LIN {X 0,Y 419.877,Z 411.6,A -85,B 0,C 180,E1 9458.97,E2 9458.97} C_VEL
LIN {X 0,Y 420.638,Z 405.188,A -85,B 0,C 180,E1 9462.43,E2 9462.43} C_VEL
LIN {X 0,Y 421.745,Z 393.076,A -85,B 0,C 180,E1 9465.832,E2 9465.832} C_VEL
LIN {X 0,Y 423.274,Z 375.401,A -85,B 0,C 180,E1 9468.881,E2 9468.881} C_VEL
LIN {X 0,Y 424.894,Z 354.463,A -85,B 0,C 180,E1 9471.197,E2 9471.197} C_VEL
LIN {X 0,Y 425.891,Z 330.735,A -85,B 0,C 180,E1 9472.858,E2 9472.858} C_VEL
LIN {X 0,Y 419.501,Z 305.694,A -85,B 0,C 180,E1 9474.153,E2 9474.153} C_VEL
LIN {X 0,Y 417.305,Z 297.81,A -85,B 0,C 180,E1 9474.446,E2 9474.446} C_VEL
LIN {X 0,Y 416.963,Z 297.81,A -85,B 0,C 180,E1 9480.442,E2 9480.442} C_VEL
LIN {X 0,Y 416.972,Z 297.81,A -85,B 0,C 180,E1 9487.211,E2 9487.211} C_VEL
LIN {X 0,Y 416.83,Z 297.81,A -85,B 0,C 180,E1 9493.591,E2 9493.591} C_VEL
LIN {X 0,Y 416.903,Z 297.81,A -85,B 0,C 180,E1 9499.474,E2 9499.474} C_VEL
LIN {X 0,Y 416.902,Z 297.81,A -85,B 0,C 180,E1 9504.594,E2 9504.594} C_VEL
LIN {X 0,Y 417.002,Z 297.81,A -85,B 0,C 180,E1 9511.922,E2 9511.922} C_VEL
LIN {X 0,Y 417.371,Z 297.81,A -85,B 0,C 180,E1 9518.79,E2 9518.79} C_VEL
LIN {X 0,Y 417.453,Z 297.81,A -85,B 0,C 180,E1 9525.329,E2 9525.329} C_VEL
LIN {X 0,Y 417.766,Z 297.81,A -85,B 0,C 180,E1 9531.679,E2 9531.679} C_VEL
LIN {X 0,Y 418.193,Z 297.81,A -85,B 0,C 180,E1 9537.919,E2 9537.919} C_VEL
LIN {X 0,Y 418.002,Z 297.81,A -85,B 0,C 180,E1 9544.128,E2 9544.128} C_VEL
LIN {X 0,Y 417.732,Z 297.81,A -85,B 0,C 180,E1 9550.393,E2 9550.393} C_VEL
LIN {X 0,Y 417.495,Z 297.81,A -85,B 0,C 180,E1 9556.794,E2 9556.794} C_VEL
LIN {X 0,Y 417.298,Z 297.81,A -85,B 0,C 180,E1 9563.426,E2 9563.426} C_VEL
LIN {X 0,Y 417.029,Z 297.81,A -85,B 0,C 180,E1 9570.423,E2 9570.423} C_VEL
LIN {X 0,Y 416.911,Z 297.81,A -85,B 0,C 180,E1 9577.96,E2 9577.96} C_VEL
LIN {X 0,Y 416.867,Z 297.81,A -85,B 0,C 180,E1 9583.616,E2 9583.616} C_VEL
LIN {X 0,Y 416.962,Z 297.81,A -85,B 0,C 180,E1 9589.446,E2 9589.446} C_VEL
LIN {X 0,Y 416.98,Z 297.81,A -85,B 0,C 180,E1 9594.618,E2 9594.618} C_VEL
LIN {X 0,Y 417.197,Z 297.81,A -85,B 0,C 180,E1 9600.595,E2 9600.595} C_VEL
LIN {X 0,Y 430.602,Z 338.236,A -85,B 0,C 180,E1 9602.059,E2 9602.059} C_VEL
LIN {X 0,Y 429.755,Z 375.538,A -85,B 0,C 180,E1 9602.915,E2 9602.915} C_VEL
LIN {X 0,Y 427.343,Z 408.592,A -85,B 0,C 180,E1 9604.471,E2 9604.471} C_VEL
LIN {X 0,Y 424.757,Z 438.385,A -85,B 0,C 180,E1 9606.719,E2 9606.719} C_VEL
LIN {X 0,Y 422.244,Z 465.016,A -85,B 0,C 180,E1 9609.607,E2 9609.607} C_VEL
LIN {X 0,Y 420.814,Z 481.386,A -85,B 0,C 180,E1 9611.972,E2 9611.972} C_VEL
LIN {X 0,Y 419.147,Z 486.865,A -85,B 0,C 180,E1 9612.877,E2 9612.877} C_VEL
LIN {X 0,Y 411.685,Z 500.03,A -85,B 0,C 180,E1 9615.497,E2 9615.497} C_VEL
LIN {X 0,Y 411.541,Z 501.128,A -85,B 0,C 180,E1 9615.76,E2 9615.76} C_VEL
LIN {X 0,Y 411.062,Z 515.83,A -85,B 0,C 180,E1 9619.957,E2 9619.957} C_VEL
LIN {X 0,Y 411.204,Z 524.231,A -85,B 0,C 180,E1 9623.679,E2 9623.679} C_VEL
LIN {X 0,Y 411.473,Z 528.984,A -85,B 0,C 180,E1 9627.898,E2 9627.898} C_VEL
LIN {X 0,Y 411.46,Z 528.901,A -85,B 0,C 180,E1 9632.101,E2 9632.101} C_VEL
LIN {X 0,Y 411.236,Z 524.018,A -85,B 0,C 180,E1 9636.319,E2 9636.319} C_VEL
LIN {X 0,Y 411.131,Z 513.977,A -85,B 0,C 180,E1 9640.574,E2 9640.574} C_VEL
LIN {X 0,Y 411.714,Z 498.169,A -85,B 0,C 180,E1 9644.865,E2 9644.865} C_VEL
LIN {X 0,Y 413.331,Z 476.598,A -85,B 0,C 180,E1 9648.901,E2 9648.901} C_VEL
LIN {X 0,Y 415.903,Z 450.804,A -85,B 0,C 180,E1 9652.327,E2 9652.327} C_VEL
LIN {X 0,Y 418.823,Z 421.694,A -85,B 0,C 180,E1 9655.045,E2 9655.045} C_VEL
LIN {X 0,Y 421.731,Z 389.924,A -85,B 0,C 180,E1 9657.003,E2 9657.003} C_VEL
LIN {X 0,Y 423.6,Z 356.055,A -85,B 0,C 180,E1 9658.183,E2 9658.183} C_VEL
LIN {X 0,Y 423.18,Z 337.903,A -85,B 0,C 180,E1 9658.562,E2 9658.562} C_VEL
LIN {X 0,Y 409.163,Z 297.81,A -85,B 0,C 180,E1 9660.29,E2 9660.29} C_VEL
LIN {X 0,Y 408.961,Z 297.81,A -85,B 0,C 180,E1 9666.183,E2 9666.183} C_VEL
LIN {X 0,Y 408.78,Z 297.81,A -85,B 0,C 180,E1 9672.431,E2 9672.431} C_VEL
LIN {X 0,Y 408.855,Z 297.81,A -85,B 0,C 180,E1 9678.384,E2 9678.384} C_VEL
LIN {X 0,Y 409.002,Z 297.81,A -85,B 0,C 180,E1 9684.259,E2 9684.259} C_VEL
LIN {X 0,Y 409.091,Z 297.81,A -85,B 0,C 180,E1 9691.36,E2 9691.36} C_VEL
LIN {X 0,Y 409.357,Z 297.81,A -85,B 0,C 180,E1 9698.383,E2 9698.383} C_VEL
LIN {X 0,Y 409.454,Z 297.81,A -85,B 0,C 180,E1 9705.063,E2 9705.063} C_VEL
LIN {X 0,Y 409.789,Z 297.81,A -85,B 0,C 180,E1 9711.543,E2 9711.543} C_VEL
LIN {X 0,Y 410.268,Z 297.81,A -85,B 0,C 180,E1 9717.905,E2 9717.905} C_VEL
LIN {X 0,Y 410.042,Z 297.81,A -85,B 0,C 180,E1 9724.234,E2 9724.234} C_VEL
LIN {X 0,Y 409.776,Z 297.81,A -85,B 0,C 180,E1 9730.624,E2 9730.624} C_VEL
LIN {X 0,Y 409.562,Z 297.81,A -85,B 0,C 180,E1 9737.157,E2 9737.157} C_VEL
LIN {X 0,Y 409.296,Z 297.81,A -85,B 0,C 180,E1 9743.941,E2 9743.941} C_VEL
LIN {X 0,Y 409.29,Z 297.81,A -85,B 0,C 180,E1 9749.69,E2 9749.69} C_VEL
LIN {X 0,Y 417.713,Z 325.419,A -85,B 0,C 180,E1 9751.453,E2 9751.453} C_VEL
LIN {X 0,Y 419.879,Z 339.663,A -85,B 0,C 180,E1 9752.561,E2 9752.561} C_VEL
LIN {X 0,Y 417.771,Z 364.033,A -85,B 0,C 180,E1 9754.786,E2 9754.786} C_VEL
LIN {X 0,Y 415.64,Z 383.831,A -85,B 0,C 180,E1 9757.541,E2 9757.541} C_VEL
LIN {X 0,Y 413.839,Z 399.154,A -85,B 0,C 180,E1 9760.783,E2 9760.783} C_VEL
LIN {X 0,Y 412.798,Z 408.597,A -85,B 0,C 180,E1 9764.011,E2 9764.011} C_VEL
LIN {X 0,Y 412.066,Z 413.417,A -85,B 0,C 180,E1 9767.11,E2 9767.11} C_VEL
LIN {X 0,Y 411.741,Z 414.45,A -85,B 0,C 180,E1 9770.344,E2 9770.344} C_VEL
LIN {X 0,Y 412.094,Z 410.619,A -85,B 0,C 180,E1 9774.135,E2 9774.135} C_VEL
LIN {X 0,Y 413.053,Z 400.769,A -85,B 0,C 180,E1 9777.935,E2 9777.935} C_VEL
LIN {X 0,Y 414.439,Z 385.481,A -85,B 0,C 180,E1 9781.372,E2 9781.372} C_VEL
LIN {X 0,Y 416.184,Z 366.055,A -85,B 0,C 180,E1 9784.209,E2 9784.209} C_VEL
LIN {X 0,Y 417.974,Z 342.348,A -85,B 0,C 180,E1 9786.502,E2 9786.502} C_VEL
LIN {X 0,Y 417.684,Z 329.677,A -85,B 0,C 180,E1 9787.428,E2 9787.428} C_VEL
LIN {X 0,Y 410.6,Z 301.996,A -85,B 0,C 180,E1 9789.12,E2 9789.12} C_VEL
LIN {X 0,Y 409.589,Z 297.81,A -85,B 0,C 180,E1 9789.347,E2 9789.347} C_VEL
LIN {X 0,Y 409.484,Z 297.81,A -85,B 0,C 180,E1 9795.052,E2 9795.052} C_VEL
LIN {X 0,Y 409.654,Z 297.81,A -85,B 0,C 180,E1 9797.865,E2 9797.865} C_VEL
LIN {X 0,Y 416.194,Z 326.756,A -85,B 0,C 180,E1 9799.049,E2 9799.049} C_VEL
LIN {X 0,Y 416.462,Z 347.34,A -85,B 0,C 180,E1 9800.353,E2 9800.353} C_VEL
LIN {X 0,Y 415.154,Z 369.979,A -85,B 0,C 180,E1 9802.561,E2 9802.561} C_VEL
LIN {X 0,Y 413.911,Z 388.142,A -85,B 0,C 180,E1 9805.295,E2 9805.295} C_VEL
LIN {X 0,Y 412.857,Z 401.668,A -85,B 0,C 180,E1 9808.43,E2 9808.43} C_VEL
LIN {X 0,Y 412.118,Z 410.765,A -85,B 0,C 180,E1 9812.099,E2 9812.099} C_VEL
LIN {X 0,Y 411.871,Z 413.347,A -85,B 0,C 180,E1 9814.203,E2 9814.203} C_VEL
LIN {X 0,Y 411.774,Z 414.218,A -85,B 0,C 180,E1 9816.312,E2 9816.312} C_VEL
LIN {X 0,Y 412.187,Z 412.205,A -85,B 0,C 180,E1 9819.483,E2 9819.483} C_VEL
LIN {X 0,Y 413.007,Z 404.681,A -85,B 0,C 180,E1 9823.17,E2 9823.17} C_VEL
LIN {X 0,Y 414.429,Z 391.258,A -85,B 0,C 180,E1 9826.664,E2 9826.664} C_VEL
LIN {X 0,Y 415.97,Z 373.143,A -85,B 0,C 180,E1 9829.606,E2 9829.606} C_VEL
LIN {X 0,Y 417.706,Z 350.966,A -85,B 0,C 180,E1 9831.907,E2 9831.907} C_VEL
LIN {X 0,Y 417.787,Z 328.647,A -85,B 0,C 180,E1 9833.411,E2 9833.411} C_VEL
LIN {X 0,Y 410.687,Z 302.83,A -85,B 0,C 180,E1 9834.689,E2 9834.689} C_VEL
LIN {X 0,Y 409.334,Z 297.81,A -85,B 0,C 180,E1 9834.959,E2 9834.959} C_VEL
LIN {X 0,Y 408.972,Z 297.81,A -85,B 0,C 180,E1 9841.908,E2 9841.908} C_VEL
LIN {X 0,Y 409.027,Z 297.81,A -85,B 0,C 180,E1 9846.177,E2 9846.177} C_VEL
LIN {X 0,Y 408.848,Z 297.81,A -85,B 0,C 180,E1 9852.403,E2 9852.403} C_VEL
LIN {X 0,Y 408.864,Z 297.81,A -85,B 0,C 180,E1 9858.35,E2 9858.35} C_VEL
LIN {X 0,Y 408.982,Z 297.81,A -85,B 0,C 180,E1 9864.265,E2 9864.265} C_VEL
LIN {X 0,Y 409.055,Z 297.81,A -85,B 0,C 180,E1 9871.327,E2 9871.327} C_VEL
LIN {X 0,Y 409.393,Z 297.81,A -85,B 0,C 180,E1 9878.356,E2 9878.356} C_VEL
LIN {X 0,Y 409.519,Z 297.81,A -85,B 0,C 180,E1 9885.038,E2 9885.038} C_VEL
LIN {X 0,Y 409.833,Z 297.81,A -85,B 0,C 180,E1 9891.517,E2 9891.517} C_VEL
LIN {X 0,Y 410.279,Z 297.81,A -85,B 0,C 180,E1 9897.879,E2 9897.879} C_VEL
LIN {X 0,Y 410.087,Z 297.81,A -85,B 0,C 180,E1 9904.207,E2 9904.207} C_VEL
LIN {X 0,Y 409.817,Z 297.81,A -85,B 0,C 180,E1 9910.596,E2 9910.596} C_VEL
LIN {X 0,Y 409.549,Z 297.81,A -85,B 0,C 180,E1 9917.13,E2 9917.13} C_VEL
LIN {X 0,Y 409.346,Z 297.81,A -85,B 0,C 180,E1 9923.909,E2 9923.909} C_VEL
LIN {X 0,Y 409.149,Z 297.81,A -85,B 0,C 180,E1 9928.636,E2 9928.636} C_VEL
LIN {X 0,Y 408.984,Z 297.81,A -85,B 0,C 180,E1 9936.166,E2 9936.166} C_VEL
LIN {X 0,Y 408.858,Z 297.81,A -85,B 0,C 180,E1 9942.425,E2 9942.425} C_VEL
LIN {X 0,Y 408.929,Z 297.81,A -85,B 0,C 180,E1 9948.377,E2 9948.377} C_VEL
LIN {X 0,Y 409.073,Z 297.81,A -85,B 0,C 180,E1 9954.227,E2 9954.227} C_VEL
LIN {X 0,Y 409.228,Z 297.81,A -85,B 0,C 180,E1 9960.114,E2 9960.114} C_VEL
LIN {X 0,Y 423.137,Z 339.386,A -85,B 0,C 180,E1 9961.671,E2 9961.671} C_VEL
LIN {X 0,Y 422.345,Z 375.855,A -85,B 0,C 180,E1 9962.552,E2 9962.552} C_VEL
LIN {X 0,Y 419.893,Z 407.972,A -85,B 0,C 180,E1 9964.097,E2 9964.097} C_VEL
LIN {X 0,Y 417.096,Z 437.994,A -85,B 0,C 180,E1 9966.407,E2 9966.407} C_VEL
LIN {X 0,Y 414.411,Z 465.492,A -85,B 0,C 180,E1 9969.483,E2 9969.483} C_VEL
LIN {X 0,Y 412.351,Z 489.264,A -85,B 0,C 180,E1 9973.25,E2 9973.25} C_VEL
LIN {X 0,Y 411.541,Z 501.128,A -85,B 0,C 180,E1 9975.76,E2 9975.76} C_VEL
LIN {X 0,Y 410.124,Z 505.338,A -85,B 0,C 180,E1 9976.814,E2 9976.814} C_VEL
LIN {X 0,Y 403.307,Z 514.812,A -85,B 0,C 180,E1 9979.819,E2 9979.819} C_VEL
LIN {X 0,Y 403.204,Z 515.557,A -85,B 0,C 180,E1 9980.112,E2 9980.112} C_VEL
LIN {X 0,Y 403.449,Z 524.741,A -85,B 0,C 180,E1 9984.634,E2 9984.634} C_VEL
LIN {X 0,Y 403.663,Z 527.883,A -85,B 0,C 180,E1 9987.857,E2 9987.857} C_VEL
LIN {X 0,Y 403.624,Z 527.805,A -85,B 0,C 180,E1 9992.142,E2 9992.142} C_VEL
LIN {X 0,Y 403.373,Z 522.91,A -85,B 0,C 180,E1 9996.443,E2 9996.443} C_VEL
LIN {X 0,Y 403.27,Z 512.845,A -85,B 0,C 180,E1 10000.783,E2 10000.783} C_VEL
LIN {X 0,Y 403.917,Z 497.006,A -85,B 0,C 180,E1 10005.159,E2 10005.159} C_VEL
LIN {X 0,Y 405.654,Z 475.39,A -85,B 0,C 180,E1 10009.273,E2 10009.273} C_VEL
LIN {X 0,Y 408.359,Z 450.086,A -85,B 0,C 180,E1 10012.696,E2 10012.696} C_VEL
LIN {X 0,Y 411.497,Z 420.27,A -85,B 0,C 180,E1 10015.523,E2 10015.523} C_VEL
LIN {X 0,Y 414.479,Z 389.251,A -85,B 0,C 180,E1 10017.457,E2 10017.457} C_VEL
LIN {X 0,Y 416.489,Z 354.953,A -85,B 0,C 180,E1 10018.663,E2 10018.663} C_VEL
LIN {X 0,Y 416.104,Z 339.832,A -85,B 0,C 180,E1 10018.992,E2 10018.992} C_VEL
LIN {X 0,Y 401.893,Z 300.98,A -85,B 0,C 180,E1 10020.724,E2 10020.724} C_VEL
LIN {X 0,Y 401.173,Z 297.81,A -85,B 0,C 180,E1 10020.968,E2 10020.968} C_VEL
LIN {X 0,Y 400.918,Z 297.81,A -85,B 0,C 180,E1 10027.796,E2 10027.796} C_VEL
LIN {X 0,Y 400.891,Z 297.81,A -85,B 0,C 180,E1 10034.359,E2 10034.359} C_VEL
LIN {X 0,Y 400.96,Z 297.81,A -85,B 0,C 180,E1 10040.24,E2 10040.24} C_VEL
LIN {X 0,Y 401.053,Z 297.81,A -85,B 0,C 180,E1 10045.869,E2 10045.869} C_VEL
LIN {X 0,Y 401.226,Z 297.81,A -85,B 0,C 180,E1 10053.186,E2 10053.186} C_VEL
LIN {X 0,Y 401.479,Z 297.81,A -85,B 0,C 180,E1 10060.242,E2 10060.242} C_VEL
LIN {X 0,Y 401.647,Z 297.81,A -85,B 0,C 180,E1 10067.638,E2 10067.638} C_VEL
LIN {X 0,Y 402.101,Z 297.81,A -85,B 0,C 180,E1 10073.549,E2 10073.549} C_VEL
LIN {X 0,Y 402.314,Z 297.81,A -85,B 0,C 180,E1 10080.013,E2 10080.013} C_VEL
LIN {X 0,Y 402.019,Z 297.81,A -85,B 0,C 180,E1 10086.479,E2 10086.479} C_VEL
LIN {X 0,Y 401.819,Z 297.81,A -85,B 0,C 180,E1 10093.036,E2 10093.036} C_VEL
LIN {X 0,Y 401.481,Z 297.81,A -85,B 0,C 180,E1 10100.01,E2 10100.01} C_VEL
LIN {X 0,Y 401.265,Z 297.81,A -85,B 0,C 180,E1 10106.841,E2 10106.841} C_VEL
LIN {X 0,Y 401.343,Z 297.81,A -85,B 0,C 180,E1 10109.099,E2 10109.099} C_VEL
LIN {X 0,Y 410.289,Z 326.49,A -85,B 0,C 180,E1 10111.007,E2 10111.007} C_VEL
LIN {X 0,Y 412.553,Z 341.624,A -85,B 0,C 180,E1 10112.228,E2 10112.228} C_VEL
LIN {X 0,Y 410.347,Z 365.317,A -85,B 0,C 180,E1 10114.463,E2 10114.463} C_VEL
LIN {X 0,Y 408.073,Z 385.161,A -85,B 0,C 180,E1 10117.289,E2 10117.289} C_VEL
LIN {X 0,Y 406.171,Z 400.332,A -85,B 0,C 180,E1 10120.576,E2 10120.576} C_VEL
LIN {X 0,Y 405.048,Z 409.833,A -85,B 0,C 180,E1 10123.913,E2 10123.913} C_VEL
LIN {X 0,Y 404.135,Z 415.11,A -85,B 0,C 180,E1 10127.772,E2 10127.772} C_VEL
LIN {X 0,Y 403.993,Z 414.846,A -85,B 0,C 180,E1 10131.688,E2 10131.688} C_VEL
LIN {X 0,Y 404.503,Z 409.804,A -85,B 0,C 180,E1 10135.182,E2 10135.182} C_VEL
LIN {X 0,Y 405.56,Z 398.95,A -85,B 0,C 180,E1 10138.875,E2 10138.875} C_VEL
LIN {X 0,Y 407.143,Z 382.739,A -85,B 0,C 180,E1 10142.243,E2 10142.243} C_VEL
LIN {X 0,Y 409.085,Z 361.576,A -85,B 0,C 180,E1 10145.114,E2 10145.114} C_VEL
LIN {X 0,Y 410.898,Z 336.576,A -85,B 0,C 180,E1 10147.321,E2 10147.321} C_VEL
LIN {X 0,Y 405.079,Z 310.18,A -85,B 0,C 180,E1 10149.132,E2 10149.132} C_VEL
LIN {X 0,Y 401.661,Z 297.81,A -85,B 0,C 180,E1 10149.818,E2 10149.818} C_VEL
LIN {X 0,Y 401.744,Z 297.81,A -85,B 0,C 180,E1 10157.539,E2 10157.539} C_VEL
LIN {X 0,Y 408.083,Z 325.34,A -85,B 0,C 180,E1 10158.629,E2 10158.629} C_VEL
LIN {X 0,Y 409.223,Z 339.175,A -85,B 0,C 180,E1 10159.443,E2 10159.443} C_VEL
LIN {X 0,Y 408.028,Z 363.678,A -85,B 0,C 180,E1 10161.494,E2 10161.494} C_VEL
LIN {X 0,Y 406.616,Z 383.649,A -85,B 0,C 180,E1 10164.143,E2 10164.143} C_VEL
LIN {X 0,Y 405.407,Z 399.18,A -85,B 0,C 180,E1 10167.334,E2 10167.334} C_VEL
LIN {X 0,Y 404.445,Z 410.014,A -85,B 0,C 180,E1 10171.07,E2 10171.07} C_VEL
LIN {X 0,Y 404.033,Z 414.49,A -85,B 0,C 180,E1 10174.284,E2 10174.284} C_VEL
LIN {X 0,Y 403.981,Z 415.285,A -85,B 0,C 180,E1 10176.435,E2 10176.435} C_VEL
LIN {X 0,Y 404.438,Z 413.177,A -85,B 0,C 180,E1 10179.666,E2 10179.666} C_VEL
LIN {X 0,Y 405.282,Z 405.709,A -85,B 0,C 180,E1 10183.366,E2 10183.366} C_VEL
LIN {X 0,Y 406.69,Z 393.245,A -85,B 0,C 180,E1 10186.712,E2 10186.712} C_VEL
LIN {X 0,Y 408.337,Z 375.967,A -85,B 0,C 180,E1 10189.664,E2 10189.664} C_VEL
LIN {X 0,Y 410.171,Z 354.486,A -85,B 0,C 180,E1 10192.034,E2 10192.034} C_VEL
LIN {X 0,Y 410.55,Z 331.066,A -85,B 0,C 180,E1 10193.692,E2 10193.692} C_VEL
LIN {X 0,Y 403.638,Z 305.412,A -85,B 0,C 180,E1 10195.035,E2 10195.035} C_VEL
LIN {X 0,Y 401.381,Z 297.81,A -85,B 0,C 180,E1 10195.373,E2 10195.373} C_VEL
LIN {X 0,Y 401.095,Z 297.81,A -85,B 0,C 180,E1 10201.784,E2 10201.784} C_VEL
LIN {X 0,Y 400.972,Z 297.81,A -85,B 0,C 180,E1 10207.762,E2 10207.762} C_VEL
LIN {X 0,Y 400.931,Z 297.81,A -85,B 0,C 180,E1 10214.327,E2 10214.327} C_VEL
LIN {X 0,Y 400.94,Z 297.81,A -85,B 0,C 180,E1 10220.203,E2 10220.203} C_VEL
LIN {X 0,Y 401.039,Z 297.81,A -85,B 0,C 180,E1 10225.874,E2 10225.874} C_VEL
LIN {X 0,Y 401.17,Z 297.81,A -85,B 0,C 180,E1 10233.152,E2 10233.152} C_VEL
LIN {X 0,Y 401.54,Z 297.81,A -85,B 0,C 180,E1 10240.216,E2 10240.216} C_VEL
LIN {X 0,Y 401.719,Z 297.81,A -85,B 0,C 180,E1 10247.597,E2 10247.597} C_VEL
LIN {X 0,Y 402.104,Z 297.81,A -85,B 0,C 180,E1 10253.522,E2 10253.522} C_VEL
LIN {X 0,Y 402.387,Z 297.81,A -85,B 0,C 180,E1 10259.987,E2 10259.987} C_VEL
LIN {X 0,Y 402.082,Z 297.81,A -85,B 0,C 180,E1 10266.451,E2 10266.451} C_VEL
LIN {X 0,Y 401.828,Z 297.81,A -85,B 0,C 180,E1 10273.008,E2 10273.008} C_VEL
LIN {X 0,Y 401.512,Z 297.81,A -85,B 0,C 180,E1 10280.019,E2 10280.019} C_VEL
LIN {X 0,Y 401.271,Z 297.81,A -85,B 0,C 180,E1 10286.811,E2 10286.811} C_VEL
LIN {X 0,Y 401.049,Z 297.81,A -85,B 0,C 180,E1 10294.345,E2 10294.345} C_VEL
LIN {X 0,Y 400.913,Z 297.81,A -85,B 0,C 180,E1 10301.167,E2 10301.167} C_VEL
LIN {X 0,Y 400.998,Z 297.81,A -85,B 0,C 180,E1 10307.362,E2 10307.362} C_VEL
LIN {X 0,Y 401.046,Z 297.81,A -85,B 0,C 180,E1 10312.984,E2 10312.984} C_VEL
LIN {X 0,Y 401.245,Z 297.81,A -85,B 0,C 180,E1 10319.635,E2 10319.635} C_VEL
LIN {X 0,Y 415.97,Z 342.223,A -85,B 0,C 180,E1 10321.318,E2 10321.318} C_VEL
LIN {X 0,Y 414.876,Z 376.886,A -85,B 0,C 180,E1 10322.207,E2 10322.207} C_VEL
LIN {X 0,Y 412.313,Z 409.139,A -85,B 0,C 180,E1 10323.827,E2 10323.827} C_VEL
LIN {X 0,Y 409.318,Z 439.73,A -85,B 0,C 180,E1 10326.29,E2 10326.29} C_VEL
LIN {X 0,Y 406.606,Z 465.95,A -85,B 0,C 180,E1 10329.355,E2 10329.355} C_VEL
LIN {X 0,Y 404.461,Z 489.292,A -85,B 0,C 180,E1 10333.193,E2 10333.193} C_VEL
LIN {X 0,Y 403.34,Z 507.849,A -85,B 0,C 180,E1 10337.577,E2 10337.577} C_VEL
LIN {X 0,Y 403.204,Z 515.557,A -85,B 0,C 180,E1 10340.112,E2 10340.112} C_VEL
LIN {X 0,Y 401.968,Z 518.366,A -85,B 0,C 180,E1 10341.282,E2 10341.282} C_VEL
LIN {X 0,Y 395.684,Z 523.681,A -85,B 0,C 180,E1 10344.572,E2 10344.572} C_VEL
LIN {X 0,Y 395.61,Z 524.049,A -85,B 0,C 180,E1 10344.887,E2 10344.887} C_VEL
LIN {X 0,Y 395.831,Z 526.779,A -85,B 0,C 180,E1 10347.815,E2 10347.815} C_VEL
LIN {X 0,Y 395.794,Z 526.71,A -85,B 0,C 180,E1 10352.184,E2 10352.184} C_VEL
LIN {X 0,Y 395.522,Z 521.807,A -85,B 0,C 180,E1 10356.572,E2 10356.572} C_VEL
LIN {X 0,Y 395.403,Z 511.719,A -85,B 0,C 180,E1 10361,E2 10361} C_VEL
LIN {X 0,Y 396.111,Z 495.854,A -85,B 0,C 180,E1 10365.465,E2 10365.465} C_VEL
LIN {X 0,Y 398.024,Z 474.011,A -85,B 0,C 180,E1 10369.692,E2 10369.692} C_VEL
LIN {X 0,Y 400.985,Z 447.763,A -85,B 0,C 180,E1 10373.269,E2 10373.269} C_VEL
LIN {X 0,Y 404.246,Z 418.855,A -85,B 0,C 180,E1 10376.015,E2 10376.015} C_VEL
LIN {X 0,Y 407.442,Z 386.585,A -85,B 0,C 180,E1 10378.022,E2 10378.022} C_VEL
LIN {X 0,Y 409.482,Z 352.456,A -85,B 0,C 180,E1 10379.194,E2 10379.194} C_VEL
LIN {X 0,Y 408.665,Z 340.268,A -85,B 0,C 180,E1 10379.497,E2 10379.497} C_VEL
LIN {X 0,Y 394.4,Z 301.933,A -85,B 0,C 180,E1 10381.297,E2 10381.297} C_VEL
LIN {X 0,Y 393.225,Z 297.81,A -85,B 0,C 180,E1 10381.622,E2 10381.622} C_VEL
LIN {X 0,Y 393.024,Z 297.81,A -85,B 0,C 180,E1 10387.901,E2 10387.901} C_VEL
LIN {X 0,Y 392.964,Z 297.81,A -85,B 0,C 180,E1 10393.725,E2 10393.725} C_VEL
LIN {X 0,Y 393.066,Z 297.81,A -85,B 0,C 180,E1 10400.156,E2 10400.156} C_VEL
LIN {X 0,Y 393.113,Z 297.81,A -85,B 0,C 180,E1 10407.616,E2 10407.616} C_VEL
LIN {X 0,Y 393.354,Z 297.81,A -85,B 0,C 180,E1 10415.054,E2 10415.054} C_VEL
LIN {X 0,Y 393.593,Z 297.81,A -85,B 0,C 180,E1 10422.153,E2 10422.153} C_VEL
LIN {X 0,Y 393.789,Z 297.81,A -85,B 0,C 180,E1 10428.967,E2 10428.967} C_VEL
LIN {X 0,Y 394.221,Z 297.81,A -85,B 0,C 180,E1 10435.623,E2 10435.623} C_VEL
LIN {X 0,Y 394.412,Z 297.81,A -85,B 0,C 180,E1 10440.014,E2 10440.014} C_VEL
LIN {X 0,Y 394.12,Z 297.81,A -85,B 0,C 180,E1 10446.61,E2 10446.61} C_VEL
LIN {X 0,Y 393.874,Z 297.81,A -85,B 0,C 180,E1 10453.304,E2 10453.304} C_VEL
LIN {X 0,Y 393.566,Z 297.81,A -85,B 0,C 180,E1 10460.202,E2 10460.202} C_VEL
LIN {X 0,Y 393.348,Z 297.81,A -85,B 0,C 180,E1 10467.426,E2 10467.426} C_VEL
LIN {X 0,Y 393.447,Z 298.356,A -85,B 0,C 180,E1 10468.51,E2 10468.51} C_VEL
LIN {X 0,Y 402.553,Z 326.374,A -85,B 0,C 180,E1 10470.447,E2 10470.447} C_VEL
LIN {X 0,Y 405.292,Z 343.205,A -85,B 0,C 180,E1 10471.852,E2 10471.852} C_VEL
LIN {X 0,Y 402.88,Z 367.271,A -85,B 0,C 180,E1 10474.2,E2 10474.2} C_VEL
LIN {X 0,Y 400.472,Z 386.904,A -85,B 0,C 180,E1 10477.095,E2 10477.095} C_VEL
LIN {X 0,Y 398.49,Z 401.676,A -85,B 0,C 180,E1 10480.411,E2 10480.411} C_VEL
LIN {X 0,Y 397.304,Z 411.07,A -85,B 0,C 180,E1 10483.811,E2 10483.811} C_VEL
LIN {X 0,Y 396.525,Z 415.487,A -85,B 0,C 180,E1 10486.765,E2 10486.765} C_VEL
LIN {X 0,Y 396.123,Z 416.783,A -85,B 0,C 180,E1 10489.654,E2 10489.654} C_VEL
LIN {X 0,Y 396.317,Z 414.453,A -85,B 0,C 180,E1 10493.116,E2 10493.116} C_VEL
LIN {X 0,Y 397.096,Z 407.305,A -85,B 0,C 180,E1 10496.75,E2 10496.75} C_VEL
LIN {X 0,Y 398.46,Z 393.887,A -85,B 0,C 180,E1 10500.508,E2 10500.508} C_VEL
LIN {X 0,Y 400.32,Z 375.839,A -85,B 0,C 180,E1 10503.712,E2 10503.712} C_VEL
LIN {X 0,Y 402.402,Z 352.061,A -85,B 0,C 180,E1 10506.474,E2 10506.474} C_VEL
LIN {X 0,Y 402.787,Z 333.301,A -85,B 0,C 180,E1 10507.999,E2 10507.999} C_VEL
LIN {X 0,Y 395.759,Z 305.27,A -85,B 0,C 180,E1 10509.862,E2 10509.862} C_VEL
LIN {X 0,Y 393.753,Z 297.81,A -85,B 0,C 180,E1 10510.262,E2 10510.262} C_VEL
LIN {X 0,Y 393.79,Z 297.81,A -85,B 0,C 180,E1 10517.168,E2 10517.168} C_VEL
LIN {X 0,Y 400.508,Z 326.609,A -85,B 0,C 180,E1 10518.343,E2 10518.343} C_VEL
LIN {X 0,Y 401.645,Z 340.367,A -85,B 0,C 180,E1 10519.173,E2 10519.173} C_VEL
LIN {X 0,Y 400.44,Z 364.205,A -85,B 0,C 180,E1 10521.195,E2 10521.195} C_VEL
LIN {X 0,Y 398.88,Z 385.191,A -85,B 0,C 180,E1 10524.029,E2 10524.029} C_VEL
LIN {X 0,Y 397.611,Z 400.552,A -85,B 0,C 180,E1 10527.282,E2 10527.282} C_VEL
LIN {X 0,Y 396.617,Z 411.25,A -85,B 0,C 180,E1 10531.091,E2 10531.091} C_VEL
LIN {X 0,Y 396.199,Z 415.632,A -85,B 0,C 180,E1 10534.369,E2 10534.369} C_VEL
LIN {X 0,Y 396.308,Z 415.898,A -85,B 0,C 180,E1 10538.005,E2 10538.005} C_VEL
LIN {X 0,Y 397.172,Z 410.434,A -85,B 0,C 180,E1 10542.062,E2 10542.062} C_VEL
LIN {X 0,Y 398.399,Z 399.835,A -85,B 0,C 180,E1 10545.657,E2 10545.657} C_VEL
LIN {X 0,Y 400.164,Z 383.7,A -85,B 0,C 180,E1 10548.958,E2 10548.958} C_VEL
LIN {X 0,Y 402.103,Z 363.489,A -85,B 0,C 180,E1 10551.608,E2 10551.608} C_VEL
LIN {X 0,Y 403.546,Z 339.665,A -85,B 0,C 180,E1 10553.592,E2 10553.592} C_VEL
LIN {X 0,Y 400.998,Z 323.128,A -85,B 0,C 180,E1 10554.638,E2 10554.638} C_VEL
LIN {X 0,Y 393.398,Z 297.81,A -85,B 0,C 180,E1 10555.841,E2 10555.841} C_VEL
LIN {X 0,Y 393.14,Z 297.81,A -85,B 0,C 180,E1 10562.505,E2 10562.505} C_VEL
LIN {X 0,Y 393.061,Z 297.81,A -85,B 0,C 180,E1 10569.818,E2 10569.818} C_VEL
LIN {X 0,Y 393.006,Z 297.81,A -85,B 0,C 180,E1 10576.848,E2 10576.848} C_VEL
LIN {X 0,Y 393.037,Z 297.81,A -85,B 0,C 180,E1 10583.733,E2 10583.733} C_VEL
LIN {X 0,Y 393.134,Z 297.81,A -85,B 0,C 180,E1 10590.05,E2 10590.05} C_VEL
LIN {X 0,Y 393.462,Z 297.81,A -85,B 0,C 180,E1 10597.433,E2 10597.433} C_VEL
LIN {X 0,Y 393.686,Z 297.81,A -85,B 0,C 180,E1 10604.422,E2 10604.422} C_VEL
LIN {X 0,Y 393.98,Z 297.81,A -85,B 0,C 180,E1 10611.173,E2 10611.173} C_VEL
LIN {X 0,Y 394.479,Z 297.81,A -85,B 0,C 180,E1 10617.794,E2 10617.794} C_VEL
LIN {X 0,Y 394.272,Z 297.81,A -85,B 0,C 180,E1 10624.376,E2 10624.376} C_VEL
LIN {X 0,Y 393.962,Z 297.81,A -85,B 0,C 180,E1 10631.028,E2 10631.028} C_VEL
LIN {X 0,Y 393.644,Z 297.81,A -85,B 0,C 180,E1 10637.845,E2 10637.845} C_VEL
LIN {X 0,Y 393.411,Z 297.81,A -85,B 0,C 180,E1 10644.942,E2 10644.942} C_VEL
LIN {X 0,Y 393.123,Z 297.81,A -85,B 0,C 180,E1 10652.491,E2 10652.491} C_VEL
LIN {X 0,Y 393.05,Z 297.81,A -85,B 0,C 180,E1 10659.839,E2 10659.839} C_VEL
LIN {X 0,Y 393.064,Z 297.81,A -85,B 0,C 180,E1 10666.82,E2 10666.82} C_VEL
LIN {X 0,Y 393.098,Z 297.81,A -85,B 0,C 180,E1 10673.699,E2 10673.699} C_VEL
LIN {X 0,Y 393.301,Z 297.81,A -85,B 0,C 180,E1 10679.138,E2 10679.138} C_VEL
LIN {X 0,Y 408.694,Z 343.948,A -85,B 0,C 180,E1 10680.932,E2 10680.932} C_VEL
LIN {X 0,Y 407.45,Z 377.92,A -85,B 0,C 180,E1 10681.856,E2 10681.856} C_VEL
LIN {X 0,Y 404.684,Z 410.629,A -85,B 0,C 180,E1 10683.583,E2 10683.583} C_VEL
LIN {X 0,Y 401.673,Z 439.556,A -85,B 0,C 180,E1 10685.985,E2 10685.985} C_VEL
LIN {X 0,Y 398.789,Z 466.374,A -85,B 0,C 180,E1 10689.222,E2 10689.222} C_VEL
LIN {X 0,Y 396.578,Z 489.31,A -85,B 0,C 180,E1 10693.133,E2 10693.133} C_VEL
LIN {X 0,Y 395.484,Z 506.608,A -85,B 0,C 180,E1 10697.326,E2 10697.326} C_VEL
LIN {X 0,Y 395.469,Z 519.533,A -85,B 0,C 180,E1 10702.123,E2 10702.123} C_VEL
LIN {X 0,Y 395.61,Z 524.049,A -85,B 0,C 180,E1 10704.887,E2 10704.887} C_VEL
LIN {X 0,Y 393.162,Z 525.74,A -85,B 0,C 180,E1 10706.747,E2 10706.747} C_VEL
LIN {X 0,Y 388.033,Z 526.228,A -85,B 0,C 180,E1 10709.573,E2 10709.573} C_VEL
LIN {X 0,Y 387.978,Z 526.243,A -85,B 0,C 180,E1 10709.9,E2 10709.9} C_VEL
LIN {X 0,Y 387.847,Z 523.79,A -85,B 0,C 180,E1 10714.462,E2 10714.462} C_VEL
LIN {X 0,Y 387.505,Z 516.306,A -85,B 0,C 180,E1 10718.961,E2 10718.961} C_VEL
LIN {X 0,Y 387.799,Z 502.428,A -85,B 0,C 180,E1 10723.788,E2 10723.788} C_VEL
LIN {X 0,Y 389.218,Z 484.115,A -85,B 0,C 180,E1 10728.068,E2 10728.068} C_VEL
LIN {X 0,Y 391.911,Z 459.878,A -85,B 0,C 180,E1 10732.049,E2 10732.049} C_VEL
LIN {X 0,Y 395.298,Z 431.94,A -85,B 0,C 180,E1 10735.274,E2 10735.274} C_VEL
LIN {X 0,Y 398.879,Z 400.973,A -85,B 0,C 180,E1 10737.684,E2 10737.684} C_VEL
LIN {X 0,Y 401.626,Z 368.375,A -85,B 0,C 180,E1 10739.237,E2 10739.237} C_VEL
LIN {X 0,Y 401.98,Z 343.234,A -85,B 0,C 180,E1 10739.922,E2 10739.922} C_VEL
LIN {X 0,Y 388.248,Z 305.961,A -85,B 0,C 180,E1 10741.721,E2 10741.721} C_VEL
LIN {X 0,Y 385.27,Z 297.81,A -85,B 0,C 180,E1 10742.278,E2 10742.278} C_VEL
LIN {X 0,Y 385.07,Z 297.81,A -85,B 0,C 180,E1 10748.828,E2 10748.828} C_VEL
LIN {X 0,Y 384.985,Z 297.81,A -85,B 0,C 180,E1 10755.145,E2 10755.145} C_VEL
LIN {X 0,Y 385.143,Z 297.81,A -85,B 0,C 180,E1 10761.591,E2 10761.591} C_VEL
LIN {X 0,Y 385.099,Z 297.81,A -85,B 0,C 180,E1 10766.746,E2 10766.746} C_VEL
LIN {X 0,Y 385.339,Z 297.81,A -85,B 0,C 180,E1 10774.247,E2 10774.247} C_VEL
LIN {X 0,Y 385.632,Z 297.81,A -85,B 0,C 180,E1 10779.904,E2 10779.904} C_VEL
LIN {X 0,Y 385.773,Z 297.81,A -85,B 0,C 180,E1 10786.44,E2 10786.44} C_VEL
LIN {X 0,Y 386.233,Z 297.81,A -85,B 0,C 180,E1 10793.283,E2 10793.283} C_VEL
LIN {X 0,Y 386.51,Z 297.81,A -85,B 0,C 180,E1 10800.014,E2 10800.014} C_VEL
LIN {X 0,Y 386.194,Z 297.81,A -85,B 0,C 180,E1 10806.746,E2 10806.746} C_VEL
LIN {X 0,Y 385.926,Z 297.81,A -85,B 0,C 180,E1 10813.583,E2 10813.583} C_VEL
LIN {X 0,Y 385.609,Z 297.81,A -85,B 0,C 180,E1 10820.637,E2 10820.637} C_VEL
LIN {X 0,Y 385.495,Z 297.81,A -85,B 0,C 180,E1 10827.81,E2 10827.81} C_VEL
LIN {X 0,Y 395.074,Z 327.2,A -85,B 0,C 180,E1 10829.93,E2 10829.93} C_VEL
LIN {X 0,Y 398.105,Z 344.041,A -85,B 0,C 180,E1 10831.404,E2 10831.404} C_VEL
LIN {X 0,Y 395.479,Z 368.644,A -85,B 0,C 180,E1 10833.854,E2 10833.854} C_VEL
LIN {X 0,Y 392.918,Z 388.5,A -85,B 0,C 180,E1 10836.868,E2 10836.868} C_VEL
LIN {X 0,Y 390.806,Z 403.091,A -85,B 0,C 180,E1 10840.25,E2 10840.25} C_VEL
LIN {X 0,Y 389.364,Z 413.379,A -85,B 0,C 180,E1 10844.256,E2 10844.256} C_VEL
LIN {X 0,Y 388.403,Z 417.797,A -85,B 0,C 180,E1 10848.665,E2 10848.665} C_VEL
LIN {X 0,Y 388.335,Z 417.135,A -85,B 0,C 180,E1 10851.558,E2 10851.558} C_VEL
LIN {X 0,Y 388.88,Z 412.041,A -85,B 0,C 180,E1 10855.302,E2 10855.302} C_VEL
LIN {X 0,Y 390.045,Z 401.298,A -85,B 0,C 180,E1 10859.125,E2 10859.125} C_VEL
LIN {X 0,Y 391.816,Z 385.022,A -85,B 0,C 180,E1 10862.665,E2 10862.665} C_VEL
LIN {X 0,Y 393.962,Z 363.67,A -85,B 0,C 180,E1 10865.685,E2 10865.685} C_VEL
LIN {X 0,Y 395.957,Z 338.05,A -85,B 0,C 180,E1 10868.041,E2 10868.041} C_VEL
LIN {X 0,Y 389.443,Z 310.528,A -85,B 0,C 180,E1 10870.035,E2 10870.035} C_VEL
LIN {X 0,Y 385.804,Z 297.81,A -85,B 0,C 180,E1 10870.731,E2 10870.731} C_VEL
LIN {X 0,Y 385.877,Z 298.601,A -85,B 0,C 180,E1 10876.825,E2 10876.825} C_VEL
LIN {X 0,Y 392.679,Z 326.393,A -85,B 0,C 180,E1 10877.963,E2 10877.963} C_VEL
LIN {X 0,Y 394.137,Z 340.563,A -85,B 0,C 180,E1 10878.828,E2 10878.828} C_VEL
LIN {X 0,Y 392.835,Z 364.708,A -85,B 0,C 180,E1 10880.884,E2 10880.884} C_VEL
LIN {X 0,Y 391.258,Z 385.075,A -85,B 0,C 180,E1 10883.634,E2 10883.634} C_VEL
LIN {X 0,Y 389.906,Z 400.886,A -85,B 0,C 180,E1 10886.95,E2 10886.95} C_VEL
LIN {X 0,Y 388.925,Z 411.378,A -85,B 0,C 180,E1 10890.556,E2 10890.556} C_VEL
LIN {X 0,Y 388.363,Z 416.773,A -85,B 0,C 180,E1 10894.458,E2 10894.458} C_VEL
LIN {X 0,Y 388.363,Z 417.425,A -85,B 0,C 180,E1 10896.695,E2 10896.695} C_VEL
LIN {X 0,Y 388.934,Z 415.124,A -85,B 0,C 180,E1 10900.056,E2 10900.056} C_VEL
LIN {X 0,Y 389.769,Z 408.673,A -85,B 0,C 180,E1 10903.433,E2 10903.433} C_VEL
LIN {X 0,Y 391.367,Z 395.956,A -85,B 0,C 180,E1 10907.098,E2 10907.098} C_VEL
LIN {X 0,Y 393.26,Z 378.677,A -85,B 0,C 180,E1 10910.203,E2 10910.203} C_VEL
LIN {X 0,Y 395.236,Z 357.776,A -85,B 0,C 180,E1 10912.631,E2 10912.631} C_VEL
LIN {X 0,Y 395.738,Z 333.882,A -85,B 0,C 180,E1 10914.425,E2 10914.425} C_VEL
LIN {X 0,Y 388.791,Z 308.185,A -85,B 0,C 180,E1 10915.867,E2 10915.867} C_VEL
LIN {X 0,Y 385.433,Z 297.81,A -85,B 0,C 180,E1 10916.346,E2 10916.346} C_VEL
LIN {X 0,Y 385.132,Z 297.81,A -85,B 0,C 180,E1 10923.267,E2 10923.267} C_VEL
LIN {X 0,Y 385.127,Z 297.81,A -85,B 0,C 180,E1 10928.823,E2 10928.823} C_VEL
LIN {X 0,Y 385.002,Z 297.81,A -85,B 0,C 180,E1 10935.108,E2 10935.108} C_VEL
LIN {X 0,Y 385.149,Z 297.81,A -85,B 0,C 180,E1 10941.592,E2 10941.592} C_VEL
LIN {X 0,Y 385.101,Z 297.81,A -85,B 0,C 180,E1 10946.712,E2 10946.712} C_VEL
LIN {X 0,Y 385.322,Z 297.81,A -85,B 0,C 180,E1 10954.255,E2 10954.255} C_VEL
LIN {X 0,Y 385.702,Z 297.81,A -85,B 0,C 180,E1 10959.879,E2 10959.879} C_VEL
LIN {X 0,Y 385.837,Z 297.81,A -85,B 0,C 180,E1 10966.414,E2 10966.414} C_VEL
LIN {X 0,Y 386.247,Z 297.81,A -85,B 0,C 180,E1 10973.255,E2 10973.255} C_VEL
LIN {X 0,Y 386.583,Z 297.81,A -85,B 0,C 180,E1 10979.986,E2 10979.986} C_VEL
LIN {X 0,Y 386.236,Z 297.81,A -85,B 0,C 180,E1 10986.717,E2 10986.717} C_VEL
LIN {X 0,Y 385.964,Z 297.81,A -85,B 0,C 180,E1 10993.553,E2 10993.553} C_VEL
LIN {X 0,Y 385.628,Z 297.81,A -85,B 0,C 180,E1 11000.606,E2 11000.606} C_VEL
LIN {X 0,Y 385.353,Z 297.81,A -85,B 0,C 180,E1 11008.013,E2 11008.013} C_VEL
LIN {X 0,Y 385.114,Z 297.81,A -85,B 0,C 180,E1 11015.981,E2 11015.981} C_VEL
LIN {X 0,Y 385.033,Z 297.81,A -85,B 0,C 180,E1 11021.871,E2 11021.871} C_VEL
LIN {X 0,Y 385.09,Z 297.81,A -85,B 0,C 180,E1 11028.228,E2 11028.228} C_VEL
LIN {X 0,Y 385.185,Z 297.81,A -85,B 0,C 180,E1 11034.01,E2 11034.01} C_VEL
LIN {X 0,Y 385.393,Z 298.459,A -85,B 0,C 180,E1 11038.637,E2 11038.637} C_VEL
LIN {X 0,Y 401.349,Z 344.758,A -85,B 0,C 180,E1 11040.512,E2 11040.512} C_VEL
LIN {X 0,Y 400.032,Z 378.442,A -85,B 0,C 180,E1 11041.474,E2 11041.474} C_VEL
LIN {X 0,Y 397.225,Z 410.067,A -85,B 0,C 180,E1 11043.189,E2 11043.189} C_VEL
LIN {X 0,Y 394.016,Z 439.476,A -85,B 0,C 180,E1 11045.688,E2 11045.688} C_VEL
LIN {X 0,Y 390.97,Z 466.775,A -85,B 0,C 180,E1 11049.082,E2 11049.082} C_VEL
LIN {X 0,Y 388.7,Z 489.301,A -85,B 0,C 180,E1 11053.072,E2 11053.072} C_VEL
LIN {X 0,Y 387.581,Z 507.331,A -85,B 0,C 180,E1 11057.684,E2 11057.684} C_VEL
LIN {X 0,Y 387.639,Z 519.395,A -85,B 0,C 180,E1 11062.514,E2 11062.514} C_VEL
LIN {X 0,Y 387.844,Z 523.831,A -85,B 0,C 180,E1 11065.536,E2 11065.536} C_VEL
LIN {X 0,Y 387.978,Z 526.243,A -85,B 0,C 180,E1 11069.9,E2 11069.9} C_VEL
LIN {X 0,Y 385.575,Z 525.71,A -85,B 0,C 180,E1 11071.799,E2 11071.799} C_VEL
LIN {X 0,Y 379.949,Z 522.211,A -85,B 0,C 180,E1 11074.964,E2 11074.964} C_VEL
LIN {X 0,Y 379.625,Z 513.948,A -85,B 0,C 180,E1 11079.725,E2 11079.725} C_VEL
LIN {X 0,Y 380.078,Z 499.239,A -85,B 0,C 180,E1 11084.66,E2 11084.66} C_VEL
LIN {X 0,Y 381.774,Z 479.921,A -85,B 0,C 180,E1 11089.031,E2 11089.031} C_VEL
LIN {X 0,Y 384.87,Z 455.058,A -85,B 0,C 180,E1 11092.998,E2 11092.998} C_VEL
LIN {X 0,Y 388.522,Z 426.596,A -85,B 0,C 180,E1 11096.172,E2 11096.172} C_VEL
LIN {X 0,Y 392.215,Z 395.388,A -85,B 0,C 180,E1 11098.487,E2 11098.487} C_VEL
LIN {X 0,Y 394.874,Z 362.758,A -85,B 0,C 180,E1 11099.929,E2 11099.929} C_VEL
LIN {X 0,Y 394.789,Z 344.436,A -85,B 0,C 180,E1 11100.44,E2 11100.44} C_VEL
LIN {X 0,Y 380.796,Z 306.722,A -85,B 0,C 180,E1 11102.352,E2 11102.352} C_VEL
LIN {X 0,Y 377.302,Z 297.81,A -85,B 0,C 180,E1 11102.896,E2 11102.896} C_VEL
LIN {X 0,Y 377.023,Z 297.81,A -85,B 0,C 180,E1 11109.82,E2 11109.82} C_VEL
LIN {X 0,Y 377.014,Z 297.81,A -85,B 0,C 180,E1 11117.141,E2 11117.141} C_VEL
LIN {X 0,Y 377.157,Z 297.81,A -85,B 0,C 180,E1 11123.148,E2 11123.148} C_VEL
LIN {X 0,Y 377.191,Z 297.81,A -85,B 0,C 180,E1 11128.678,E2 11128.678} C_VEL
LIN {X 0,Y 377.402,Z 297.81,A -85,B 0,C 180,E1 11133.923,E2 11133.923} C_VEL
LIN {X 0,Y 377.607,Z 297.81,A -85,B 0,C 180,E1 11138.935,E2 11138.935} C_VEL
LIN {X 0,Y 377.828,Z 297.81,A -85,B 0,C 180,E1 11146.149,E2 11146.149} C_VEL
LIN {X 0,Y 378.306,Z 297.81,A -85,B 0,C 180,E1 11153.141,E2 11153.141} C_VEL
LIN {X 0,Y 378.607,Z 297.81,A -85,B 0,C 180,E1 11160.014,E2 11160.014} C_VEL
LIN {X 0,Y 378.282,Z 297.81,A -85,B 0,C 180,E1 11166.888,E2 11166.888} C_VEL
LIN {X 0,Y 377.978,Z 297.81,A -85,B 0,C 180,E1 11173.874,E2 11173.874} C_VEL
LIN {X 0,Y 377.64,Z 297.81,A -85,B 0,C 180,E1 11181.093,E2 11181.093} C_VEL
LIN {X 0,Y 377.536,Z 297.838,A -85,B 0,C 180,E1 11187.14,E2 11187.14} C_VEL
LIN {X 0,Y 387.394,Z 327.083,A -85,B 0,C 180,E1 11189.314,E2 11189.314} C_VEL
LIN {X 0,Y 390.817,Z 346.403,A -85,B 0,C 180,E1 11191.055,E2 11191.055} C_VEL
LIN {X 0,Y 387.954,Z 371.428,A -85,B 0,C 180,E1 11193.67,E2 11193.67} C_VEL
LIN {X 0,Y 385.166,Z 391.488,A -85,B 0,C 180,E1 11196.913,E2 11196.913} C_VEL
LIN {X 0,Y 382.935,Z 406.052,A -85,B 0,C 180,E1 11200.557,E2 11200.557} C_VEL
LIN {X 0,Y 381.457,Z 415.32,A -85,B 0,C 180,E1 11204.598,E2 11204.598} C_VEL
LIN {X 0,Y 380.57,Z 418.987,A -85,B 0,C 180,E1 11208.907,E2 11208.907} C_VEL
LIN {X 0,Y 380.593,Z 417.433,A -85,B 0,C 180,E1 11212.49,E2 11212.49} C_VEL
LIN {X 0,Y 381.33,Z 411.003,A -85,B 0,C 180,E1 11216.359,E2 11216.359} C_VEL
LIN {X 0,Y 382.693,Z 398.919,A -85,B 0,C 180,E1 11220.199,E2 11220.199} C_VEL
LIN {X 0,Y 384.622,Z 381.68,A -85,B 0,C 180,E1 11223.653,E2 11223.653} C_VEL
LIN {X 0,Y 386.941,Z 358.876,A -85,B 0,C 180,E1 11226.641,E2 11226.641} C_VEL
LIN {X 0,Y 388.205,Z 338.274,A -85,B 0,C 180,E1 11228.479,E2 11228.479} C_VEL
LIN {X 0,Y 381.597,Z 310.676,A -85,B 0,C 180,E1 11230.51,E2 11230.51} C_VEL
LIN {X 0,Y 377.903,Z 297.81,A -85,B 0,C 180,E1 11231.22,E2 11231.22} C_VEL
LIN {X 0,Y 377.889,Z 297.81,A -85,B 0,C 180,E1 11236.399,E2 11236.399} C_VEL
LIN {X 0,Y 385.153,Z 327.765,A -85,B 0,C 180,E1 11237.66,E2 11237.66} C_VEL
LIN {X 0,Y 386.51,Z 342.896,A -85,B 0,C 180,E1 11238.614,E2 11238.614} C_VEL
LIN {X 0,Y 385.164,Z 366.496,A -85,B 0,C 180,E1 11240.7,E2 11240.7} C_VEL
LIN {X 0,Y 383.524,Z 386.612,A -85,B 0,C 180,E1 11243.506,E2 11243.506} C_VEL
LIN {X 0,Y 382.114,Z 402.251,A -85,B 0,C 180,E1 11246.888,E2 11246.888} C_VEL
LIN {X 0,Y 381.093,Z 412.612,A -85,B 0,C 180,E1 11250.568,E2 11250.568} C_VEL
LIN {X 0,Y 380.53,Z 417.914,A -85,B 0,C 180,E1 11254.55,E2 11254.55} C_VEL
LIN {X 0,Y 380.608,Z 418.352,A -85,B 0,C 180,E1 11257.496,E2 11257.496} C_VEL
LIN {X 0,Y 381.437,Z 414.42,A -85,B 0,C 180,E1 11261.409,E2 11261.409} C_VEL
LIN {X 0,Y 382.613,Z 405.608,A -85,B 0,C 180,E1 11265.082,E2 11265.082} C_VEL
LIN {X 0,Y 384.566,Z 390.593,A -85,B 0,C 180,E1 11268.71,E2 11268.71} C_VEL
LIN {X 0,Y 386.636,Z 371.703,A -85,B 0,C 180,E1 11271.614,E2 11271.614} C_VEL
LIN {X 0,Y 388.554,Z 348.216,A -85,B 0,C 180,E1 11273.911,E2 11273.911} C_VEL
LIN {X 0,Y 388.237,Z 334.786,A -85,B 0,C 180,E1 11274.851,E2 11274.851} C_VEL
LIN {X 0,Y 381.339,Z 309.623,A -85,B 0,C 180,E1 11276.312,E2 11276.312} C_VEL
LIN {X 0,Y 377.471,Z 297.81,A -85,B 0,C 180,E1 11276.842,E2 11276.842} C_VEL
LIN {X 0,Y 377.198,Z 297.81,A -85,B 0,C 180,E1 11284.062,E2 11284.062} C_VEL
LIN {X 0,Y 377.08,Z 297.81,A -85,B 0,C 180,E1 11290.482,E2 11290.482} C_VEL
LIN {X 0,Y 377.03,Z 297.81,A -85,B 0,C 180,E1 11297.104,E2 11297.104} C_VEL
LIN {X 0,Y 377.179,Z 297.81,A -85,B 0,C 180,E1 11303.145,E2 11303.145} C_VEL
LIN {X 0,Y 377.185,Z 297.81,A -85,B 0,C 180,E1 11308.644,E2 11308.644} C_VEL
LIN {X 0,Y 377.375,Z 297.81,A -85,B 0,C 180,E1 11313.889,E2 11313.889} C_VEL
LIN {X 0,Y 377.657,Z 297.81,A -85,B 0,C 180,E1 11318.908,E2 11318.908} C_VEL
LIN {X 0,Y 377.892,Z 297.81,A -85,B 0,C 180,E1 11326.122,E2 11326.122} C_VEL
LIN {X 0,Y 378.325,Z 297.81,A -85,B 0,C 180,E1 11333.113,E2 11333.113} C_VEL
LIN {X 0,Y 378.68,Z 297.81,A -85,B 0,C 180,E1 11339.986,E2 11339.986} C_VEL
LIN {X 0,Y 378.317,Z 297.81,A -85,B 0,C 180,E1 11346.858,E2 11346.858} C_VEL
LIN {X 0,Y 378.01,Z 297.81,A -85,B 0,C 180,E1 11353.844,E2 11353.844} C_VEL
LIN {X 0,Y 377.661,Z 297.81,A -85,B 0,C 180,E1 11361.061,E2 11361.061} C_VEL
LIN {X 0,Y 377.355,Z 297.81,A -85,B 0,C 180,E1 11368.661,E2 11368.661} C_VEL
LIN {X 0,Y 377.169,Z 297.81,A -85,B 0,C 180,E1 11374.048,E2 11374.048} C_VEL
LIN {X 0,Y 377.06,Z 297.81,A -85,B 0,C 180,E1 11380.501,E2 11380.501} C_VEL
LIN {X 0,Y 377.075,Z 297.81,A -85,B 0,C 180,E1 11387.131,E2 11387.131} C_VEL
LIN {X 0,Y 377.234,Z 297.81,A -85,B 0,C 180,E1 11393.128,E2 11393.128} C_VEL
LIN {X 0,Y 377.429,Z 297.81,A -85,B 0,C 180,E1 11398.039,E2 11398.039} C_VEL
LIN {X 0,Y 393.928,Z 345.832,A -85,B 0,C 180,E1 11400.075,E2 11400.075} C_VEL
LIN {X 0,Y 392.481,Z 380.99,A -85,B 0,C 180,E1 11401.159,E2 11401.159} C_VEL
LIN {X 0,Y 389.468,Z 413.009,A -85,B 0,C 180,E1 11403.034,E2 11403.034} C_VEL
LIN {X 0,Y 386.017,Z 442.833,A -85,B 0,C 180,E1 11405.766,E2 11405.766} C_VEL
LIN {X 0,Y 382.926,Z 468.88,A -85,B 0,C 180,E1 11409.227,E2 11409.227} C_VEL
LIN {X 0,Y 380.673,Z 490.718,A -85,B 0,C 180,E1 11413.329,E2 11413.329} C_VEL
LIN {X 0,Y 379.687,Z 507.957,A -85,B 0,C 180,E1 11418.03,E2 11418.03} C_VEL
LIN {X 0,Y 379.808,Z 518.618,A -85,B 0,C 180,E1 11422.58,E2 11422.58} C_VEL
LIN {X 0,Y 380.01,Z 522.699,A -85,B 0,C 180,E1 11425.444,E2 11425.444} C_VEL
LIN {X 0,Y 380.169,Z 525.167,A -85,B 0,C 180,E1 11429.999,E2 11429.999} C_VEL
LIN {X 0,Y 380.012,Z 522.701,A -85,B 0,C 180,E1 11434.554,E2 11434.554} C_VEL
LIN {X 0,Y 379.949,Z 522.211,A -85,B 0,C 180,E1 11434.964,E2 11434.964} C_VEL
LIN {X 0,Y 377.24,Z 519.368,A -85,B 0,C 180,E1 11436.864,E2 11436.864} C_VEL
LIN {X 0,Y 371.838,Z 513.507,A -85,B 0,C 180,E1 11439.659,E2 11439.659} C_VEL
LIN {X 0,Y 371.751,Z 512.742,A -85,B 0,C 180,E1 11439.978,E2 11439.978} C_VEL
LIN {X 0,Y 372.289,Z 498.123,A -85,B 0,C 180,E1 11444.974,E2 11444.974} C_VEL
LIN {X 0,Y 374.105,Z 478.799,A -85,B 0,C 180,E1 11449.436,E2 11449.436} C_VEL
LIN {X 0,Y 377.318,Z 454.719,A -85,B 0,C 180,E1 11453.369,E2 11453.369} C_VEL
LIN {X 0,Y 381.157,Z 426.508,A -85,B 0,C 180,E1 11456.601,E2 11456.601} C_VEL
LIN {X 0,Y 385.101,Z 394.918,A -85,B 0,C 180,E1 11459.006,E2 11459.006} C_VEL
LIN {X 0,Y 387.859,Z 362.845,A -85,B 0,C 180,E1 11460.457,E2 11460.457} C_VEL
LIN {X 0,Y 387.695,Z 345.732,A -85,B 0,C 180,E1 11460.97,E2 11460.97} C_VEL
LIN {X 0,Y 374.095,Z 309.506,A -85,B 0,C 180,E1 11462.903,E2 11462.903} C_VEL
LIN {X 0,Y 369.299,Z 297.81,A -85,B 0,C 180,E1 11463.644,E2 11463.644} C_VEL
LIN {X 0,Y 369.062,Z 297.81,A -85,B 0,C 180,E1 11470.858,E2 11470.858} C_VEL
LIN {X 0,Y 369.098,Z 297.81,A -85,B 0,C 180,E1 11477.382,E2 11477.382} C_VEL
LIN {X 0,Y 369.153,Z 297.81,A -85,B 0,C 180,E1 11484.838,E2 11484.838} C_VEL
LIN {X 0,Y 369.309,Z 297.81,A -85,B 0,C 180,E1 11490.654,E2 11490.654} C_VEL
LIN {X 0,Y 369.526,Z 297.81,A -85,B 0,C 180,E1 11495.913,E2 11495.913} C_VEL
LIN {X 0,Y 369.822,Z 297.81,A -85,B 0,C 180,E1 11503.419,E2 11503.419} C_VEL
LIN {X 0,Y 370.125,Z 297.81,A -85,B 0,C 180,E1 11510.629,E2 11510.629} C_VEL
LIN {X 0,Y 370.74,Z 297.81,A -85,B 0,C 180,E1 11517.682,E2 11517.682} C_VEL
LIN {X 0,Y 370.498,Z 297.81,A -85,B 0,C 180,E1 11524.687,E2 11524.687} C_VEL
LIN {X 0,Y 370.142,Z 297.81,A -85,B 0,C 180,E1 11531.925,E2 11531.925} C_VEL
LIN {X 0,Y 369.789,Z 297.81,A -85,B 0,C 180,E1 11539.07,E2 11539.07} C_VEL
LIN {X 0,Y 369.595,Z 297.817,A -85,B 0,C 180,E1 11546.401,E2 11546.401} C_VEL
LIN {X 0,Y 379.703,Z 327.028,A -85,B 0,C 180,E1 11548.662,E2 11548.662} C_VEL
LIN {X 0,Y 383.675,Z 347.5,A -85,B 0,C 180,E1 11550.587,E2 11550.587} C_VEL
LIN {X 0,Y 380.662,Z 372.494,A -85,B 0,C 180,E1 11553.251,E2 11553.251} C_VEL
LIN {X 0,Y 377.688,Z 392.635,A -85,B 0,C 180,E1 11556.578,E2 11556.578} C_VEL
LIN {X 0,Y 375.345,Z 406.851,A -85,B 0,C 180,E1 11560.196,E2 11560.196} C_VEL
LIN {X 0,Y 373.725,Z 416.435,A -85,B 0,C 180,E1 11564.429,E2 11564.429} C_VEL
LIN {X 0,Y 373.112,Z 419.13,A -85,B 0,C 180,E1 11566.741,E2 11566.741} C_VEL
LIN {X 0,Y 372.674,Z 419.937,A -85,B 0,C 180,E1 11570.319,E2 11570.319} C_VEL
LIN {X 0,Y 372.99,Z 416.615,A -85,B 0,C 180,E1 11574.039,E2 11574.039} C_VEL
LIN {X 0,Y 374.049,Z 408.221,A -85,B 0,C 180,E1 11577.937,E2 11577.937} C_VEL
LIN {X 0,Y 375.667,Z 394.479,A -85,B 0,C 180,E1 11581.68,E2 11581.68} C_VEL
LIN {X 0,Y 377.853,Z 375.334,A -85,B 0,C 180,E1 11585.041,E2 11585.041} C_VEL
LIN {X 0,Y 380.118,Z 352.705,A -85,B 0,C 180,E1 11587.691,E2 11587.691} C_VEL
LIN {X 0,Y 380.467,Z 338.398,A -85,B 0,C 180,E1 11588.935,E2 11588.935} C_VEL
LIN {X 0,Y 373.786,Z 310.798,A -85,B 0,C 180,E1 11591.006,E2 11591.006} C_VEL
LIN {X 0,Y 369.916,Z 297.81,A -85,B 0,C 180,E1 11591.725,E2 11591.725} C_VEL
LIN {X 0,Y 369.946,Z 297.931,A -85,B 0,C 180,E1 11596.016,E2 11596.016} C_VEL
LIN {X 0,Y 377.281,Z 327.35,A -85,B 0,C 180,E1 11597.239,E2 11597.239} C_VEL
LIN {X 0,Y 379,Z 343.235,A -85,B 0,C 180,E1 11598.253,E2 11598.253} C_VEL
LIN {X 0,Y 377.615,Z 366.979,A -85,B 0,C 180,E1 11600.368,E2 11600.368} C_VEL
LIN {X 0,Y 375.965,Z 386.473,A -85,B 0,C 180,E1 11603.085,E2 11603.085} C_VEL
LIN {X 0,Y 374.43,Z 402.577,A -85,B 0,C 180,E1 11606.535,E2 11606.535} C_VEL
LIN {X 0,Y 373.273,Z 413.842,A -85,B 0,C 180,E1 11610.58,E2 11610.58} C_VEL
LIN {X 0,Y 372.714,Z 419.049,A -85,B 0,C 180,E1 11614.645,E2 11614.645} C_VEL
LIN {X 0,Y 372.732,Z 419.568,A -85,B 0,C 180,E1 11616.977,E2 11616.977} C_VEL
LIN {X 0,Y 373.409,Z 417.081,A -85,B 0,C 180,E1 11620.478,E2 11620.478} C_VEL
LIN {X 0,Y 374.605,Z 409.064,A -85,B 0,C 180,E1 11624.507,E2 11624.507} C_VEL
LIN {X 0,Y 376.448,Z 396.122,A -85,B 0,C 180,E1 11628.1,E2 11628.1} C_VEL
LIN {X 0,Y 378.617,Z 377.676,A -85,B 0,C 180,E1 11631.327,E2 11631.327} C_VEL
LIN {X 0,Y 380.849,Z 354.856,A -85,B 0,C 180,E1 11633.855,E2 11633.855} C_VEL
LIN {X 0,Y 380.891,Z 336.375,A -85,B 0,C 180,E1 11635.246,E2 11635.246} C_VEL
LIN {X 0,Y 374.056,Z 311.277,A -85,B 0,C 180,E1 11636.76,E2 11636.76} C_VEL
LIN {X 0,Y 369.516,Z 297.81,A -85,B 0,C 180,E1 11637.408,E2 11637.408} C_VEL
LIN {X 0,Y 369.188,Z 297.81,A -85,B 0,C 180,E1 11645.14,E2 11645.14} C_VEL
LIN {X 0,Y 369.121,Z 297.81,A -85,B 0,C 180,E1 11652.597,E2 11652.597} C_VEL
LIN {X 0,Y 369.122,Z 297.81,A -85,B 0,C 180,E1 11659.128,E2 11659.128} C_VEL
LIN {X 0,Y 369.178,Z 297.81,A -85,B 0,C 180,E1 11665.074,E2 11665.074} C_VEL
LIN {X 0,Y 369.267,Z 297.81,A -85,B 0,C 180,E1 11670.617,E2 11670.617} C_VEL
LIN {X 0,Y 369.541,Z 297.81,A -85,B 0,C 180,E1 11675.882,E2 11675.882} C_VEL
LIN {X 0,Y 369.799,Z 297.81,A -85,B 0,C 180,E1 11680.931,E2 11680.931} C_VEL
LIN {X 0,Y 370.06,Z 297.81,A -85,B 0,C 180,E1 11688.22,E2 11688.22} C_VEL
LIN {X 0,Y 370.509,Z 297.81,A -85,B 0,C 180,E1 11695.313,E2 11695.313} C_VEL
LIN {X 0,Y 370.801,Z 297.81,A -85,B 0,C 180,E1 11699.985,E2 11699.985} C_VEL
LIN {X 0,Y 370.387,Z 297.81,A -85,B 0,C 180,E1 11707.006,E2 11707.006} C_VEL
LIN {X 0,Y 370.084,Z 297.81,A -85,B 0,C 180,E1 11714.146,E2 11714.146} C_VEL
LIN {X 0,Y 369.719,Z 297.81,A -85,B 0,C 180,E1 11721.536,E2 11721.536} C_VEL
LIN {X 0,Y 369.485,Z 297.81,A -85,B 0,C 180,E1 11726.68,E2 11726.68} C_VEL
LIN {X 0,Y 369.285,Z 297.81,A -85,B 0,C 180,E1 11732.071,E2 11732.071} C_VEL
LIN {X 0,Y 369.102,Z 297.81,A -85,B 0,C 180,E1 11739.033,E2 11739.033} C_VEL
LIN {X 0,Y 369.157,Z 297.81,A -85,B 0,C 180,E1 11745.979,E2 11745.979} C_VEL
LIN {X 0,Y 369.229,Z 297.81,A -85,B 0,C 180,E1 11752.19,E2 11752.19} C_VEL
LIN {X 0,Y 369.444,Z 297.81,A -85,B 0,C 180,E1 11757.483,E2 11757.483} C_VEL
LIN {X 0,Y 386.722,Z 347.732,A -85,B 0,C 180,E1 11759.667,E2 11759.667} C_VEL
LIN {X 0,Y 385.079,Z 381.423,A -85,B 0,C 180,E1 11760.756,E2 11760.756} C_VEL
LIN {X 0,Y 381.937,Z 413.36,A -85,B 0,C 180,E1 11762.683,E2 11762.683} C_VEL
LIN {X 0,Y 378.424,Z 442.272,A -85,B 0,C 180,E1 11765.404,E2 11765.404} C_VEL
LIN {X 0,Y 375.335,Z 467.313,A -85,B 0,C 180,E1 11768.786,E2 11768.786} C_VEL
LIN {X 0,Y 372.919,Z 489.496,A -85,B 0,C 180,E1 11773.011,E2 11773.011} C_VEL
LIN {X 0,Y 371.849,Z 505.938,A -85,B 0,C 180,E1 11777.531,E2 11777.531} C_VEL
LIN {X 0,Y 371.925,Z 517.441,A -85,B 0,C 180,E1 11782.422,E2 11782.422} C_VEL
LIN {X 0,Y 372.166,Z 521.562,A -85,B 0,C 180,E1 11785.348,E2 11785.348} C_VEL
LIN {X 0,Y 372.345,Z 524.062,A -85,B 0,C 180,E1 11789.999,E2 11789.999} C_VEL
LIN {X 0,Y 372.128,Z 521.303,A -85,B 0,C 180,E1 11794.915,E2 11794.915} C_VEL
LIN {X 0,Y 371.751,Z 512.742,A -85,B 0,C 180,E1 11799.978,E2 11799.978} C_VEL
LIN {X 0,Y 369.289,Z 507.938,A -85,B 0,C 180,E1 11801.829,E2 11801.829} C_VEL
LIN {X 0,Y 364.375,Z 499.626,A -85,B 0,C 180,E1 11804.542,E2 11804.542} C_VEL
LIN {X 0,Y 364.373,Z 498.577,A -85,B 0,C 180,E1 11804.848,E2 11804.848} C_VEL
LIN {X 0,Y 366.252,Z 479.214,A -85,B 0,C 180,E1 11809.557,E2 11809.557} C_VEL
LIN {X 0,Y 369.644,Z 455.34,A -85,B 0,C 180,E1 11813.624,E2 11813.624} C_VEL
LIN {X 0,Y 373.564,Z 428.09,A -85,B 0,C 180,E1 11816.889,E2 11816.889} C_VEL
LIN {X 0,Y 377.592,Z 397.737,A -85,B 0,C 180,E1 11819.335,E2 11819.335} C_VEL
LIN {X 0,Y 380.75,Z 364.853,A -85,B 0,C 180,E1 11820.937,E2 11820.937} C_VEL
LIN {X 0,Y 380.891,Z 347.862,A -85,B 0,C 180,E1 11821.481,E2 11821.481} C_VEL
LIN {X 0,Y 367.075,Z 311.239,A -85,B 0,C 180,E1 11823.536,E2 11823.536} C_VEL
LIN {X 0,Y 361.289,Z 297.81,A -85,B 0,C 180,E1 11824.575,E2 11824.575} C_VEL
LIN {X 0,Y 361.139,Z 297.81,A -85,B 0,C 180,E1 11831.954,E2 11831.954} C_VEL
LIN {X 0,Y 361.198,Z 297.81,A -85,B 0,C 180,E1 11838.762,E2 11838.762} C_VEL
LIN {X 0,Y 361.177,Z 297.81,A -85,B 0,C 180,E1 11844.22,E2 11844.22} C_VEL
LIN {X 0,Y 361.371,Z 297.81,A -85,B 0,C 180,E1 11851.27,E2 11851.27} C_VEL
LIN {X 0,Y 361.679,Z 297.81,A -85,B 0,C 180,E1 11857.96,E2 11857.96} C_VEL
LIN {X 0,Y 361.953,Z 297.81,A -85,B 0,C 180,E1 11865.529,E2 11865.529} C_VEL
LIN {X 0,Y 362.446,Z 297.81,A -85,B 0,C 180,E1 11872.84,E2 11872.84} C_VEL
LIN {X 0,Y 362.827,Z 297.81,A -85,B 0,C 180,E1 11880.015,E2 11880.015} C_VEL
LIN {X 0,Y 362.442,Z 297.81,A -85,B 0,C 180,E1 11887.19,E2 11887.19} C_VEL
LIN {X 0,Y 362.085,Z 297.81,A -85,B 0,C 180,E1 11894.496,E2 11894.496} C_VEL
LIN {X 0,Y 361.721,Z 297.81,A -85,B 0,C 180,E1 11902.069,E2 11902.069} C_VEL
LIN {X 0,Y 361.676,Z 298.27,A -85,B 0,C 180,E1 11905.626,E2 11905.626} C_VEL
LIN {X 0,Y 371.983,Z 326.646,A -85,B 0,C 180,E1 11907.948,E2 11907.948} C_VEL
LIN {X 0,Y 376.455,Z 349.45,A -85,B 0,C 180,E1 11910.17,E2 11910.17} C_VEL
LIN {X 0,Y 373.318,Z 374.03,A -85,B 0,C 180,E1 11912.881,E2 11912.881} C_VEL
LIN {X 0,Y 370.158,Z 394.085,A -85,B 0,C 180,E1 11916.287,E2 11916.287} C_VEL
LIN {X 0,Y 367.722,Z 408.056,A -85,B 0,C 180,E1 11919.942,E2 11919.942} C_VEL
LIN {X 0,Y 366.274,Z 416.252,A -85,B 0,C 180,E1 11923.444,E2 11923.444} C_VEL
LIN {X 0,Y 365.637,Z 419.122,A -85,B 0,C 180,E1 11925.446,E2 11925.446} C_VEL
LIN {X 0,Y 364.978,Z 421.178,A -85,B 0,C 180,E1 11928.585,E2 11928.585} C_VEL
LIN {X 0,Y 365.011,Z 418.965,A -85,B 0,C 180,E1 11933.125,E2 11933.125} C_VEL
LIN {X 0,Y 365.938,Z 411.756,A -85,B 0,C 180,E1 11937.138,E2 11937.138} C_VEL
LIN {X 0,Y 367.5,Z 399.403,A -85,B 0,C 180,E1 11940.991,E2 11940.991} C_VEL
LIN {X 0,Y 369.64,Z 381.53,A -85,B 0,C 180,E1 11944.542,E2 11944.542} C_VEL
LIN {X 0,Y 372.121,Z 359.384,A -85,B 0,C 180,E1 11947.468,E2 11947.468} C_VEL
LIN {X 0,Y 373.012,Z 340.038,A -85,B 0,C 180,E1 11949.27,E2 11949.27} C_VEL
LIN {X 0,Y 366.631,Z 313.283,A -85,B 0,C 180,E1 11951.376,E2 11951.376} C_VEL
LIN {X 0,Y 362.009,Z 297.81,A -85,B 0,C 180,E1 11952.332,E2 11952.332} C_VEL
LIN {X 0,Y 361.999,Z 297.965,A -85,B 0,C 180,E1 11955.593,E2 11955.593} C_VEL
LIN {X 0,Y 369.738,Z 328.514,A -85,B 0,C 180,E1 11956.897,E2 11956.897} C_VEL
LIN {X 0,Y 371.453,Z 344.892,A -85,B 0,C 180,E1 11957.974,E2 11957.974} C_VEL
LIN {X 0,Y 369.939,Z 368.752,A -85,B 0,C 180,E1 11960.166,E2 11960.166} C_VEL
LIN {X 0,Y 368.067,Z 389.66,A -85,B 0,C 180,E1 11963.232,E2 11963.232} C_VEL
LIN {X 0,Y 366.539,Z 404.974,A -85,B 0,C 180,E1 11966.756,E2 11966.756} C_VEL
LIN {X 0,Y 365.459,Z 415.07,A -85,B 0,C 180,E1 11970.592,E2 11970.592} C_VEL
LIN {X 0,Y 364.882,Z 420.178,A -85,B 0,C 180,E1 11974.745,E2 11974.745} C_VEL
LIN {X 0,Y 364.925,Z 420.639,A -85,B 0,C 180,E1 11977.127,E2 11977.127} C_VEL
LIN {X 0,Y 365.663,Z 418.06,A -85,B 0,C 180,E1 11980.703,E2 11980.703} C_VEL
LIN {X 0,Y 366.909,Z 410.21,A -85,B 0,C 180,E1 11984.711,E2 11984.711} C_VEL
LIN {X 0,Y 368.922,Z 396.83,A -85,B 0,C 180,E1 11988.482,E2 11988.482} C_VEL
LIN {X 0,Y 371.254,Z 378.183,A -85,B 0,C 180,E1 11991.771,E2 11991.771} C_VEL
LIN {X 0,Y 373.607,Z 355.014,A -85,B 0,C 180,E1 11994.347,E2 11994.347} C_VEL
LIN {X 0,Y 373.595,Z 338.123,A -85,B 0,C 180,E1 11995.644,E2 11995.644} C_VEL
LIN {X 0,Y 366.635,Z 312.614,A -85,B 0,C 180,E1 11997.246,E2 11997.246} C_VEL
LIN {X 0,Y 361.556,Z 297.81,A -85,B 0,C 180,E1 11998.076,E2 11998.076} C_VEL
LIN {X 0,Y 361.207,Z 297.81,A -85,B 0,C 180,E1 12005.795,E2 12005.795} C_VEL
LIN {X 0,Y 361.214,Z 297.81,A -85,B 0,C 180,E1 12011.945,E2 12011.945} C_VEL
LIN {X 0,Y 361.222,Z 297.81,A -85,B 0,C 180,E1 12018.76,E2 12018.76} C_VEL
LIN {X 0,Y 361.188,Z 297.81,A -85,B 0,C 180,E1 12024.184,E2 12024.184} C_VEL
LIN {X 0,Y 361.327,Z 297.81,A -85,B 0,C 180,E1 12031.286,E2 12031.286} C_VEL
LIN {X 0,Y 361.722,Z 297.81,A -85,B 0,C 180,E1 12037.931,E2 12037.931} C_VEL
LIN {X 0,Y 362.016,Z 297.81,A -85,B 0,C 180,E1 12045.501,E2 12045.501} C_VEL
LIN {X 0,Y 362.454,Z 297.81,A -85,B 0,C 180,E1 12053.092,E2 12053.092} C_VEL
LIN {X 0,Y 362.898,Z 297.81,A -85,B 0,C 180,E1 12059.985,E2 12059.985} C_VEL
LIN {X 0,Y 362.472,Z 297.81,A -85,B 0,C 180,E1 12067.16,E2 12067.16} C_VEL
LIN {X 0,Y 362.124,Z 297.81,A -85,B 0,C 180,E1 12074.464,E2 12074.464} C_VEL
LIN {X 0,Y 361.736,Z 297.81,A -85,B 0,C 180,E1 12082.036,E2 12082.036} C_VEL
LIN {X 0,Y 361.405,Z 297.81,A -85,B 0,C 180,E1 12088.737,E2 12088.737} C_VEL
LIN {X 0,Y 361.181,Z 297.81,A -85,B 0,C 180,E1 12095.78,E2 12095.78} C_VEL
LIN {X 0,Y 361.192,Z 297.81,A -85,B 0,C 180,E1 12101.929,E2 12101.929} C_VEL
LIN {X 0,Y 361.263,Z 297.81,A -85,B 0,C 180,E1 12108.731,E2 12108.731} C_VEL
LIN {X 0,Y 361.474,Z 297.81,A -85,B 0,C 180,E1 12116.583,E2 12116.583} C_VEL
LIN {X 0,Y 361.525,Z 298.574,A -85,B 0,C 180,E1 12116.949,E2 12116.949} C_VEL
LIN {X 0,Y 379.423,Z 349.283,A -85,B 0,C 180,E1 12119.232,E2 12119.232} C_VEL
LIN {X 0,Y 377.6,Z 382.981,A -85,B 0,C 180,E1 12120.403,E2 12120.403} C_VEL
LIN {X 0,Y 374.336,Z 414.532,A -85,B 0,C 180,E1 12122.401,E2 12122.401} C_VEL
LIN {X 0,Y 370.547,Z 444.227,A -85,B 0,C 180,E1 12125.328,E2 12125.328} C_VEL
LIN {X 0,Y 367.272,Z 469.357,A -85,B 0,C 180,E1 12128.929,E2 12128.929} C_VEL
LIN {X 0,Y 364.94,Z 490.312,A -85,B 0,C 180,E1 12133.175,E2 12133.175} C_VEL
LIN {X 0,Y 363.927,Z 506.858,A -85,B 0,C 180,E1 12138.034,E2 12138.034} C_VEL
LIN {X 0,Y 364.152,Z 517.266,A -85,B 0,C 180,E1 12142.858,E2 12142.858} C_VEL
LIN {X 0,Y 364.482,Z 522.33,A -85,B 0,C 180,E1 12147.627,E2 12147.627} C_VEL
LIN {X 0,Y 364.446,Z 522.331,A -85,B 0,C 180,E1 12152.372,E2 12152.372} C_VEL
LIN {X 0,Y 364.111,Z 517.426,A -85,B 0,C 180,E1 12157.141,E2 12157.141} C_VEL
LIN {X 0,Y 363.951,Z 506.246,A -85,B 0,C 180,E1 12162.346,E2 12162.346} C_VEL
LIN {X 0,Y 364.373,Z 498.577,A -85,B 0,C 180,E1 12164.848,E2 12164.848} C_VEL
LIN {X 0,Y 363.493,Z 494.354,A -85,B 0,C 180,E1 12166.047,E2 12166.047} C_VEL
LIN {X 0,Y 358.219,Z 481.684,A -85,B 0,C 180,E1 12169.227,E2 12169.227} C_VEL
LIN {X 0,Y 358.295,Z 480.392,A -85,B 0,C 180,E1 12169.514,E2 12169.514} C_VEL
LIN {X 0,Y 361.882,Z 456.297,A -85,B 0,C 180,E1 12173.834,E2 12173.834} C_VEL
LIN {X 0,Y 366.069,Z 428.948,A -85,B 0,C 180,E1 12177.253,E2 12177.253} C_VEL
LIN {X 0,Y 370.453,Z 397.936,A -85,B 0,C 180,E1 12179.848,E2 12179.848} C_VEL
LIN {X 0,Y 373.8,Z 365.262,A -85,B 0,C 180,E1 12181.502,E2 12181.502} C_VEL
LIN {X 0,Y 374.172,Z 350.136,A -85,B 0,C 180,E1 12182.012,E2 12182.012} C_VEL
LIN {X 0,Y 360.717,Z 314.552,A -85,B 0,C 180,E1 12184.104,E2 12184.104} C_VEL
LIN {X 0,Y 353.32,Z 297.81,A -85,B 0,C 180,E1 12185.344,E2 12185.344} C_VEL
LIN {X 0,Y 353.146,Z 297.81,A -85,B 0,C 180,E1 12193.131,E2 12193.131} C_VEL
LIN {X 0,Y 353.24,Z 297.81,A -85,B 0,C 180,E1 12200.257,E2 12200.257} C_VEL
LIN {X 0,Y 353.288,Z 297.81,A -85,B 0,C 180,E1 12206.288,E2 12206.288} C_VEL
LIN {X 0,Y 353.507,Z 297.81,A -85,B 0,C 180,E1 12213.689,E2 12213.689} C_VEL
LIN {X 0,Y 353.821,Z 297.81,A -85,B 0,C 180,E1 12220.066,E2 12220.066} C_VEL
LIN {X 0,Y 354.163,Z 297.81,A -85,B 0,C 180,E1 12227.715,E2 12227.715} C_VEL
LIN {X 0,Y 354.665,Z 297.81,A -85,B 0,C 180,E1 12235.134,E2 12235.134} C_VEL
LIN {X 0,Y 354.93,Z 297.81,A -85,B 0,C 180,E1 12240.015,E2 12240.015} C_VEL
LIN {X 0,Y 354.509,Z 297.81,A -85,B 0,C 180,E1 12247.352,E2 12247.352} C_VEL
LIN {X 0,Y 354.161,Z 297.81,A -85,B 0,C 180,E1 12254.828,E2 12254.828} C_VEL
LIN {X 0,Y 353.785,Z 297.81,A -85,B 0,C 180,E1 12262.591,E2 12262.591} C_VEL
LIN {X 0,Y 353.758,Z 297.81,A -85,B 0,C 180,E1 12264.766,E2 12264.766} C_VEL
LIN {X 0,Y 364.534,Z 327.137,A -85,B 0,C 180,E1 12267.272,E2 12267.272} C_VEL
LIN {X 0,Y 369.423,Z 350.481,A -85,B 0,C 180,E1 12269.65,E2 12269.65} C_VEL
LIN {X 0,Y 366.069,Z 375.122,A -85,B 0,C 180,E1 12272.422,E2 12272.422} C_VEL
LIN {X 0,Y 362.77,Z 394.818,A -85,B 0,C 180,E1 12275.831,E2 12275.831} C_VEL
LIN {X 0,Y 360.213,Z 408.547,A -85,B 0,C 180,E1 12279.443,E2 12279.443} C_VEL
LIN {X 0,Y 358.545,Z 417.54,A -85,B 0,C 180,E1 12283.326,E2 12283.326} C_VEL
LIN {X 0,Y 357.325,Z 421.979,A -85,B 0,C 180,E1 12287.494,E2 12287.494} C_VEL
LIN {X 0,Y 357.096,Z 421.03,A -85,B 0,C 180,E1 12292.172,E2 12292.172} C_VEL
LIN {X 0,Y 358.03,Z 413.979,A -85,B 0,C 180,E1 12296.777,E2 12296.777} C_VEL
LIN {X 0,Y 359.675,Z 401.084,A -85,B 0,C 180,E1 12301.036,E2 12301.036} C_VEL
LIN {X 0,Y 361.969,Z 383.289,A -85,B 0,C 180,E1 12304.711,E2 12304.711} C_VEL
LIN {X 0,Y 364.642,Z 360.469,A -85,B 0,C 180,E1 12307.815,E2 12307.815} C_VEL
LIN {X 0,Y 365.58,Z 341.666,A -85,B 0,C 180,E1 12309.619,E2 12309.619} C_VEL
LIN {X 0,Y 359.123,Z 314.271,A -85,B 0,C 180,E1 12311.843,E2 12311.843} C_VEL
LIN {X 0,Y 354.09,Z 297.81,A -85,B 0,C 180,E1 12312.906,E2 12312.906} C_VEL
LIN {X 0,Y 354.063,Z 297.81,A -85,B 0,C 180,E1 12315.127,E2 12315.127} C_VEL
LIN {X 0,Y 362.165,Z 329.58,A -85,B 0,C 180,E1 12316.535,E2 12316.535} C_VEL
LIN {X 0,Y 363.95,Z 345.599,A -85,B 0,C 180,E1 12317.614,E2 12317.614} C_VEL
LIN {X 0,Y 362.384,Z 369.236,A -85,B 0,C 180,E1 12319.807,E2 12319.807} C_VEL
LIN {X 0,Y 360.512,Z 389.529,A -85,B 0,C 180,E1 12322.787,E2 12322.787} C_VEL
LIN {X 0,Y 358.875,Z 405.292,A -85,B 0,C 180,E1 12326.385,E2 12326.385} C_VEL
LIN {X 0,Y 357.644,Z 416.297,A -85,B 0,C 180,E1 12330.605,E2 12330.605} C_VEL
LIN {X 0,Y 357.059,Z 421.296,A -85,B 0,C 180,E1 12334.849,E2 12334.849} C_VEL
LIN {X 0,Y 357.117,Z 421.712,A -85,B 0,C 180,E1 12337.283,E2 12337.283} C_VEL
LIN {X 0,Y 357.902,Z 419.042,A -85,B 0,C 180,E1 12340.938,E2 12340.938} C_VEL
LIN {X 0,Y 359.314,Z 410.729,A -85,B 0,C 180,E1 12345.155,E2 12345.155} C_VEL
LIN {X 0,Y 361.413,Z 397.527,A -85,B 0,C 180,E1 12348.88,E2 12348.88} C_VEL
LIN {X 0,Y 363.926,Z 378.663,A -85,B 0,C 180,E1 12352.233,E2 12352.233} C_VEL
LIN {X 0,Y 366.29,Z 356.38,A -85,B 0,C 180,E1 12354.748,E2 12354.748} C_VEL
LIN {X 0,Y 366.573,Z 341.03,A -85,B 0,C 180,E1 12355.965,E2 12355.965} C_VEL
LIN {X 0,Y 359.826,Z 315.634,A -85,B 0,C 180,E1 12357.66,E2 12357.66} C_VEL
LIN {X 0,Y 353.585,Z 297.81,A -85,B 0,C 180,E1 12358.567,E2 12358.567} C_VEL
LIN {X 0,Y 353.277,Z 297.81,A -85,B 0,C 180,E1 12366.728,E2 12366.728} C_VEL
LIN {X 0,Y 353.187,Z 297.81,A -85,B 0,C 180,E1 12373.396,E2 12373.396} C_VEL
LIN {X 0,Y 353.236,Z 297.81,A -85,B 0,C 180,E1 12380.26,E2 12380.26} C_VEL
LIN {X 0,Y 353.288,Z 297.81,A -85,B 0,C 180,E1 12386.251,E2 12386.251} C_VEL
LIN {X 0,Y 353.588,Z 297.81,A -85,B 0,C 180,E1 12394.72,E2 12394.72} C_VEL
LIN {X 0,Y 353.883,Z 297.81,A -85,B 0,C 180,E1 12400.037,E2 12400.037} C_VEL
LIN {X 0,Y 354.217,Z 297.81,A -85,B 0,C 180,E1 12407.686,E2 12407.686} C_VEL
LIN {X 0,Y 354.687,Z 297.81,A -85,B 0,C 180,E1 12415.103,E2 12415.103} C_VEL
LIN {X 0,Y 354.999,Z 297.81,A -85,B 0,C 180,E1 12419.985,E2 12419.985} C_VEL
LIN {X 0,Y 354.539,Z 297.81,A -85,B 0,C 180,E1 12427.321,E2 12427.321} C_VEL
LIN {X 0,Y 354.191,Z 297.81,A -85,B 0,C 180,E1 12434.795,E2 12434.795} C_VEL
LIN {X 0,Y 353.787,Z 297.81,A -85,B 0,C 180,E1 12442.558,E2 12442.558} C_VEL
LIN {X 0,Y 353.516,Z 297.81,A -85,B 0,C 180,E1 12447.988,E2 12447.988} C_VEL
LIN {X 0,Y 353.295,Z 297.81,A -85,B 0,C 180,E1 12455.753,E2 12455.753} C_VEL
LIN {X 0,Y 353.198,Z 297.81,A -85,B 0,C 180,E1 12463.422,E2 12463.422} C_VEL
LIN {X 0,Y 353.303,Z 297.81,A -85,B 0,C 180,E1 12470.225,E2 12470.225} C_VEL
LIN {X 0,Y 353.53,Z 297.81,A -85,B 0,C 180,E1 12476.296,E2 12476.296} C_VEL
LIN {X 0,Y 372.168,Z 350.983,A -85,B 0,C 180,E1 12478.785,E2 12478.785} C_VEL
LIN {X 0,Y 370.16,Z 384.179,A -85,B 0,C 180,E1 12480.016,E2 12480.016} C_VEL
LIN {X 0,Y 366.75,Z 415.443,A -85,B 0,C 180,E1 12482.092,E2 12482.092} C_VEL
LIN {X 0,Y 362.807,Z 444.727,A -85,B 0,C 180,E1 12485.094,E2 12485.094} C_VEL
LIN {X 0,Y 359.438,Z 469.513,A -85,B 0,C 180,E1 12488.77,E2 12488.77} C_VEL
LIN {X 0,Y 356.938,Z 491.402,A -85,B 0,C 180,E1 12493.419,E2 12493.419} C_VEL
LIN {X 0,Y 356.047,Z 507.203,A -85,B 0,C 180,E1 12498.385,E2 12498.385} C_VEL
LIN {X 0,Y 356.274,Z 516.076,A -85,B 0,C 180,E1 12502.699,E2 12502.699} C_VEL
LIN {X 0,Y 356.658,Z 521.215,A -85,B 0,C 180,E1 12507.574,E2 12507.574} C_VEL
LIN {X 0,Y 356.626,Z 521.241,A -85,B 0,C 180,E1 12512.424,E2 12512.424} C_VEL
LIN {X 0,Y 356.246,Z 516.335,A -85,B 0,C 180,E1 12517.3,E2 12517.3} C_VEL
LIN {X 0,Y 356.047,Z 506.202,A -85,B 0,C 180,E1 12522.234,E2 12522.234} C_VEL
LIN {X 0,Y 357.172,Z 490.268,A -85,B 0,C 180,E1 12527.201,E2 12527.201} C_VEL
LIN {X 0,Y 358.295,Z 480.392,A -85,B 0,C 180,E1 12529.514,E2 12529.514} C_VEL
LIN {X 0,Y 356.004,Z 469.984,A -85,B 0,C 180,E1 12531.748,E2 12531.748} C_VEL
LIN {X 0,Y 353.93,Z 458.46,A -85,B 0,C 180,E1 12533.858,E2 12533.858} C_VEL
LIN {X 0,Y 358.322,Z 431.792,A -85,B 0,C 180,E1 12537.426,E2 12537.426} C_VEL
LIN {X 0,Y 362.994,Z 401.151,A -85,B 0,C 180,E1 12540.183,E2 12540.183} C_VEL
LIN {X 0,Y 366.568,Z 369.55,A -85,B 0,C 180,E1 12541.934,E2 12541.934} C_VEL
LIN {X 0,Y 367.133,Z 351.374,A -85,B 0,C 180,E1 12542.607,E2 12542.607} C_VEL
LIN {X 0,Y 354.031,Z 316.938,A -85,B 0,C 180,E1 12544.756,E2 12544.756} C_VEL
LIN {X 0,Y 345.361,Z 297.81,A -85,B 0,C 180,E1 12546.245,E2 12546.245} C_VEL
LIN {X 0,Y 345.158,Z 297.81,A -85,B 0,C 180,E1 12554.386,E2 12554.386} C_VEL
LIN {X 0,Y 345.22,Z 297.81,A -85,B 0,C 180,E1 12561.886,E2 12561.886} C_VEL
LIN {X 0,Y 345.411,Z 297.81,A -85,B 0,C 180,E1 12568.4,E2 12568.4} C_VEL
LIN {X 0,Y 345.711,Z 297.81,A -85,B 0,C 180,E1 12576.437,E2 12576.437} C_VEL
LIN {X 0,Y 345.981,Z 297.81,A -85,B 0,C 180,E1 12583.641,E2 12583.641} C_VEL
LIN {X 0,Y 346.326,Z 297.81,A -85,B 0,C 180,E1 12589.978,E2 12589.978} C_VEL
LIN {X 0,Y 347.029,Z 297.81,A -85,B 0,C 180,E1 12597.523,E2 12597.523} C_VEL
LIN {X 0,Y 346.758,Z 297.81,A -85,B 0,C 180,E1 12605.009,E2 12605.009} C_VEL
LIN {X 0,Y 346.343,Z 297.81,A -85,B 0,C 180,E1 12612.599,E2 12612.599} C_VEL
LIN {X 0,Y 345.923,Z 297.81,A -85,B 0,C 180,E1 12620.442,E2 12620.442} C_VEL
LIN {X 0,Y 345.873,Z 298.496,A -85,B 0,C 180,E1 12623.895,E2 12623.895} C_VEL
LIN {X 0,Y 357.035,Z 327.415,A -85,B 0,C 180,E1 12626.532,E2 12626.532} C_VEL
LIN {X 0,Y 362.236,Z 350.43,A -85,B 0,C 180,E1 12628.978,E2 12628.978} C_VEL
LIN {X 0,Y 359.128,Z 374.344,A -85,B 0,C 180,E1 12631.682,E2 12631.682} C_VEL
LIN {X 0,Y 355.738,Z 393.956,A -85,B 0,C 180,E1 12635,E2 12635} C_VEL
LIN {X 0,Y 352.671,Z 409.524,A -85,B 0,C 180,E1 12639.08,E2 12639.08} C_VEL
LIN {X 0,Y 350.657,Z 419.348,A -85,B 0,C 180,E1 12643.537,E2 12643.537} C_VEL
LIN {X 0,Y 349.574,Z 423.016,A -85,B 0,C 180,E1 12647.234,E2 12647.234} C_VEL
LIN {X 0,Y 349.234,Z 422.881,A -85,B 0,C 180,E1 12651.083,E2 12651.083} C_VEL
LIN {X 0,Y 349.936,Z 417.069,A -85,B 0,C 180,E1 12655.904,E2 12655.904} C_VEL
LIN {X 0,Y 351.413,Z 406.067,A -85,B 0,C 180,E1 12660.137,E2 12660.137} C_VEL
LIN {X 0,Y 353.677,Z 389.816,A -85,B 0,C 180,E1 12664.007,E2 12664.007} C_VEL
LIN {X 0,Y 356.38,Z 368.176,A -85,B 0,C 180,E1 12667.376,E2 12667.376} C_VEL
LIN {X 0,Y 358.179,Z 343.553,A -85,B 0,C 180,E1 12669.949,E2 12669.949} C_VEL
LIN {X 0,Y 351.659,Z 315.763,A -85,B 0,C 180,E1 12672.303,E2 12672.303} C_VEL
LIN {X 0,Y 346.184,Z 297.81,A -85,B 0,C 180,E1 12673.493,E2 12673.493} C_VEL
LIN {X 0,Y 346.156,Z 297.81,A -85,B 0,C 180,E1 12674.684,E2 12674.684} C_VEL
LIN {X 0,Y 354.447,Z 329.751,A -85,B 0,C 180,E1 12676.104,E2 12676.104} C_VEL
LIN {X 0,Y 356.41,Z 347.411,A -85,B 0,C 180,E1 12677.323,E2 12677.323} C_VEL
LIN {X 0,Y 354.741,Z 370.988,A -85,B 0,C 180,E1 12679.585,E2 12679.585} C_VEL
LIN {X 0,Y 352.813,Z 391.047,A -85,B 0,C 180,E1 12682.629,E2 12682.629} C_VEL
LIN {X 0,Y 351.084,Z 406.648,A -85,B 0,C 180,E1 12686.304,E2 12686.304} C_VEL
LIN {X 0,Y 349.824,Z 417.523,A -85,B 0,C 180,E1 12690.619,E2 12690.619} C_VEL
LIN {X 0,Y 349.227,Z 422.412,A -85,B 0,C 180,E1 12694.958,E2 12694.958} C_VEL
LIN {X 0,Y 349.325,Z 422.782,A -85,B 0,C 180,E1 12697.447,E2 12697.447} C_VEL
LIN {X 0,Y 350.158,Z 420.025,A -85,B 0,C 180,E1 12701.183,E2 12701.183} C_VEL
LIN {X 0,Y 351.729,Z 411.417,A -85,B 0,C 180,E1 12705.554,E2 12705.554} C_VEL
LIN {X 0,Y 353.914,Z 398.229,A -85,B 0,C 180,E1 12709.296,E2 12709.296} C_VEL
LIN {X 0,Y 356.452,Z 380.243,A -85,B 0,C 180,E1 12712.561,E2 12712.561} C_VEL
LIN {X 0,Y 359.005,Z 357.625,A -85,B 0,C 180,E1 12715.178,E2 12715.178} C_VEL
LIN {X 0,Y 359.002,Z 341.298,A -85,B 0,C 180,E1 12716.517,E2 12716.517} C_VEL
LIN {X 0,Y 352.145,Z 315.975,A -85,B 0,C 180,E1 12718.239,E2 12718.239} C_VEL
LIN {X 0,Y 345.608,Z 297.81,A -85,B 0,C 180,E1 12719.207,E2 12719.207} C_VEL
LIN {X 0,Y 345.361,Z 297.81,A -85,B 0,C 180,E1 12724.613,E2 12724.613} C_VEL
LIN {X 0,Y 345.184,Z 297.81,A -85,B 0,C 180,E1 12731.973,E2 12731.973} C_VEL
LIN {X 0,Y 345.196,Z 297.81,A -85,B 0,C 180,E1 12739.004,E2 12739.004} C_VEL
LIN {X 0,Y 345.381,Z 297.81,A -85,B 0,C 180,E1 12746.113,E2 12746.113} C_VEL
LIN {X 0,Y 345.642,Z 297.81,A -85,B 0,C 180,E1 12754.096,E2 12754.096} C_VEL
LIN {X 0,Y 345.93,Z 297.81,A -85,B 0,C 180,E1 12759.558,E2 12759.558} C_VEL
LIN {X 0,Y 346.268,Z 297.81,A -85,B 0,C 180,E1 12767.398,E2 12767.398} C_VEL
LIN {X 0,Y 346.77,Z 297.81,A -85,B 0,C 180,E1 12774.991,E2 12774.991} C_VEL
LIN {X 0,Y 347.076,Z 297.81,A -85,B 0,C 180,E1 12780.236,E2 12780.236} C_VEL
LIN {X 0,Y 346.626,Z 297.81,A -85,B 0,C 180,E1 12787.489,E2 12787.489} C_VEL
LIN {X 0,Y 346.222,Z 297.81,A -85,B 0,C 180,E1 12795.144,E2 12795.144} C_VEL
LIN {X 0,Y 345.794,Z 297.81,A -85,B 0,C 180,E1 12803.109,E2 12803.109} C_VEL
LIN {X 0,Y 345.475,Z 297.81,A -85,B 0,C 180,E1 12809.122,E2 12809.122} C_VEL
LIN {X 0,Y 345.373,Z 297.81,A -85,B 0,C 180,E1 12814.593,E2 12814.593} C_VEL
LIN {X 0,Y 345.2,Z 297.81,A -85,B 0,C 180,E1 12822,E2 12822} C_VEL
LIN {X 0,Y 345.245,Z 297.81,A -85,B 0,C 180,E1 12829.032,E2 12829.032} C_VEL
LIN {X 0,Y 345.553,Z 297.81,A -85,B 0,C 180,E1 12835.675,E2 12835.675} C_VEL
LIN {X 0,Y 364.933,Z 352.856,A -85,B 0,C 180,E1 12838.339,E2 12838.339} C_VEL
LIN {X 0,Y 362.607,Z 386.637,A -85,B 0,C 180,E1 12839.683,E2 12839.683} C_VEL
LIN {X 0,Y 358.928,Z 417.955,A -85,B 0,C 180,E1 12841.907,E2 12841.907} C_VEL
LIN {X 0,Y 354.894,Z 446.587,A -85,B 0,C 180,E1 12845.029,E2 12845.029} C_VEL
LIN {X 0,Y 351.37,Z 471.277,A -85,B 0,C 180,E1 12848.919,E2 12848.919} C_VEL
LIN {X 0,Y 348.994,Z 492.334,A -85,B 0,C 180,E1 12853.676,E2 12853.676} C_VEL
LIN {X 0,Y 348.165,Z 507.508,A -85,B 0,C 180,E1 12858.752,E2 12858.752} C_VEL
LIN {X 0,Y 348.509,Z 516.661,A -85,B 0,C 180,E1 12863.786,E2 12863.786} C_VEL
LIN {X 0,Y 348.823,Z 520.096,A -85,B 0,C 180,E1 12867.52,E2 12867.52} C_VEL
LIN {X 0,Y 348.792,Z 520.149,A -85,B 0,C 180,E1 12872.479,E2 12872.479} C_VEL
LIN {X 0,Y 348.374,Z 515.252,A -85,B 0,C 180,E1 12877.466,E2 12877.466} C_VEL
LIN {X 0,Y 348.22,Z 504.088,A -85,B 0,C 180,E1 12882.91,E2 12882.91} C_VEL
LIN {X 0,Y 349.662,Z 487.531,A -85,B 0,C 180,E1 12888.012,E2 12888.012} C_VEL
LIN {X 0,Y 352.717,Z 465.706,A -85,B 0,C 180,E1 12892.645,E2 12892.645} C_VEL
LIN {X 0,Y 353.93,Z 458.46,A -85,B 0,C 180,E1 12893.858,E2 12893.858} C_VEL
LIN {X 0,Y 352.179,Z 446.262,A -85,B 0,C 180,E1 12895.873,E2 12895.873} C_VEL
LIN {X 0,Y 350.776,Z 433.111,A -85,B 0,C 180,E1 12897.761,E2 12897.761} C_VEL
LIN {X 0,Y 355.653,Z 403.027,A -85,B 0,C 180,E1 12900.606,E2 12900.606} C_VEL
LIN {X 0,Y 359.527,Z 371.741,A -85,B 0,C 180,E1 12902.459,E2 12902.459} C_VEL
LIN {X 0,Y 360.225,Z 352.985,A -85,B 0,C 180,E1 12903.213,E2 12903.213} C_VEL
LIN {X 0,Y 347.583,Z 319.564,A -85,B 0,C 180,E1 12905.42,E2 12905.42} C_VEL
LIN {X 0,Y 337.342,Z 297.81,A -85,B 0,C 180,E1 12907.274,E2 12907.274} C_VEL
LIN {X 0,Y 337.246,Z 297.81,A -85,B 0,C 180,E1 12914.303,E2 12914.303} C_VEL
LIN {X 0,Y 337.268,Z 297.81,A -85,B 0,C 180,E1 12921.235,E2 12921.235} C_VEL
LIN {X 0,Y 337.488,Z 297.81,A -85,B 0,C 180,E1 12928.16,E2 12928.16} C_VEL
LIN {X 0,Y 337.805,Z 297.81,A -85,B 0,C 180,E1 12936.311,E2 12936.311} C_VEL
LIN {X 0,Y 337.984,Z 297.81,A -85,B 0,C 180,E1 12941.805,E2 12941.805} C_VEL
LIN {X 0,Y 338.385,Z 297.81,A -85,B 0,C 180,E1 12949.741,E2 12949.741} C_VEL
LIN {X 0,Y 339.11,Z 297.81,A -85,B 0,C 180,E1 12957.465,E2 12957.465} C_VEL
LIN {X 0,Y 338.831,Z 297.81,A -85,B 0,C 180,E1 12965.126,E2 12965.126} C_VEL
LIN {X 0,Y 338.389,Z 297.81,A -85,B 0,C 180,E1 12972.9,E2 12972.9} C_VEL
LIN {X 0,Y 337.957,Z 297.81,A -85,B 0,C 180,E1 12980.946,E2 12980.946} C_VEL
LIN {X 0,Y 337.974,Z 298.533,A -85,B 0,C 180,E1 12982.928,E2 12982.928} C_VEL
LIN {X 0,Y 349.608,Z 327.798,A -85,B 0,C 180,E1 12985.76,E2 12985.76} C_VEL
LIN {X 0,Y 355.026,Z 351.667,A -85,B 0,C 180,E1 12988.393,E2 12988.393} C_VEL
LIN {X 0,Y 351.86,Z 376.141,A -85,B 0,C 180,E1 12991.269,E2 12991.269} C_VEL
LIN {X 0,Y 348.199,Z 395.961,A -85,B 0,C 180,E1 12994.766,E2 12994.766} C_VEL
LIN {X 0,Y 345.202,Z 410.325,A -85,B 0,C 180,E1 12998.635,E2 12998.635} C_VEL
LIN {X 0,Y 343.091,Z 419.909,A -85,B 0,C 180,E1 13002.935,E2 13002.935} C_VEL
LIN {X 0,Y 342.344,Z 422.739,A -85,B 0,C 180,E1 13005.151,E2 13005.151} C_VEL
LIN {X 0,Y 341.526,Z 424.562,A -85,B 0,C 180,E1 13008.714,E2 13008.714} C_VEL
LIN {X 0,Y 341.518,Z 422.765,A -85,B 0,C 180,E1 13012.715,E2 13012.715} C_VEL
LIN {X 0,Y 342.6,Z 414.956,A -85,B 0,C 180,E1 13017.505,E2 13017.505} C_VEL
LIN {X 0,Y 344.416,Z 402.143,A -85,B 0,C 180,E1 13021.738,E2 13021.738} C_VEL
LIN {X 0,Y 346.96,Z 383.812,A -85,B 0,C 180,E1 13025.568,E2 13025.568} C_VEL
LIN {X 0,Y 349.816,Z 361.331,A -85,B 0,C 180,E1 13028.684,E2 13028.684} C_VEL
LIN {X 0,Y 350.779,Z 345.298,A -85,B 0,C 180,E1 13030.305,E2 13030.305} C_VEL
LIN {X 0,Y 344.42,Z 317.798,A -85,B 0,C 180,E1 13032.732,E2 13032.732} C_VEL
LIN {X 0,Y 338.279,Z 297.81,A -85,B 0,C 180,E1 13034.065,E2 13034.065} C_VEL
LIN {X 0,Y 347.41,Z 333.287,A -85,B 0,C 180,E1 13035.872,E2 13035.872} C_VEL
LIN {X 0,Y 348.882,Z 348.796,A -85,B 0,C 180,E1 13036.986,E2 13036.986} C_VEL
LIN {X 0,Y 347.095,Z 372.699,A -85,B 0,C 180,E1 13039.353,E2 13039.353} C_VEL
LIN {X 0,Y 345.08,Z 392.565,A -85,B 0,C 180,E1 13042.463,E2 13042.463} C_VEL
LIN {X 0,Y 343.292,Z 408.003,A -85,B 0,C 180,E1 13046.22,E2 13046.22} C_VEL
LIN {X 0,Y 342.011,Z 418.748,A -85,B 0,C 180,E1 13050.633,E2 13050.633} C_VEL
LIN {X 0,Y 341.413,Z 423.526,A -85,B 0,C 180,E1 13055.072,E2 13055.072} C_VEL
LIN {X 0,Y 341.523,Z 423.853,A -85,B 0,C 180,E1 13057.618,E2 13057.618} C_VEL
LIN {X 0,Y 342.409,Z 421.009,A -85,B 0,C 180,E1 13061.439,E2 13061.439} C_VEL
LIN {X 0,Y 344.109,Z 412.276,A -85,B 0,C 180,E1 13065.908,E2 13065.908} C_VEL
LIN {X 0,Y 346.454,Z 398.931,A -85,B 0,C 180,E1 13069.729,E2 13069.729} C_VEL
LIN {X 0,Y 349.17,Z 380.727,A -85,B 0,C 180,E1 13073.058,E2 13073.058} C_VEL
LIN {X 0,Y 351.762,Z 358.233,A -85,B 0,C 180,E1 13075.689,E2 13075.689} C_VEL
LIN {X 0,Y 352.007,Z 344.246,A -85,B 0,C 180,E1 13076.858,E2 13076.858} C_VEL
LIN {X 0,Y 345.523,Z 319.421,A -85,B 0,C 180,E1 13078.663,E2 13078.663} C_VEL
LIN {X 0,Y 337.615,Z 297.81,A -85,B 0,C 180,E1 13079.973,E2 13079.973} C_VEL
LIN {X 0,Y 337.294,Z 297.81,A -85,B 0,C 180,E1 13086.332,E2 13086.332} C_VEL
LIN {X 0,Y 337.255,Z 297.81,A -85,B 0,C 180,E1 13094.258,E2 13094.258} C_VEL
LIN {X 0,Y 337.253,Z 297.81,A -85,B 0,C 180,E1 13101.192,E2 13101.192} C_VEL
LIN {X 0,Y 337.493,Z 297.81,A -85,B 0,C 180,E1 13108.161,E2 13108.161} C_VEL
LIN {X 0,Y 337.831,Z 297.81,A -85,B 0,C 180,E1 13116.278,E2 13116.278} C_VEL
LIN {X 0,Y 338.047,Z 297.81,A -85,B 0,C 180,E1 13121.774,E2 13121.774} C_VEL
LIN {X 0,Y 338.436,Z 297.81,A -85,B 0,C 180,E1 13129.71,E2 13129.71} C_VEL
LIN {X 0,Y 339.125,Z 297.81,A -85,B 0,C 180,E1 13137.434,E2 13137.434} C_VEL
LIN {X 0,Y 339.036,Z 297.81,A -85,B 0,C 180,E1 13142.535,E2 13142.535} C_VEL
LIN {X 0,Y 338.527,Z 297.81,A -85,B 0,C 180,E1 13150.255,E2 13150.255} C_VEL
LIN {X 0,Y 338.088,Z 297.81,A -85,B 0,C 180,E1 13158.19,E2 13158.19} C_VEL
LIN {X 0,Y 337.857,Z 297.81,A -85,B 0,C 180,E1 13163.685,E2 13163.685} C_VEL
LIN {X 0,Y 337.534,Z 297.81,A -85,B 0,C 180,E1 13171.85,E2 13171.85} C_VEL
LIN {X 0,Y 337.273,Z 297.81,A -85,B 0,C 180,E1 13178.764,E2 13178.764} C_VEL
LIN {X 0,Y 337.311,Z 297.81,A -85,B 0,C 180,E1 13185.686,E2 13185.686} C_VEL
LIN {X 0,Y 337.422,Z 297.81,A -85,B 0,C 180,E1 13193.584,E2 13193.584} C_VEL
LIN {X 0,Y 337.548,Z 297.81,A -85,B 0,C 180,E1 13194.997,E2 13194.997} C_VEL
LIN {X 0,Y 357.706,Z 355.488,A -85,B 0,C 180,E1 13197.92,E2 13197.92} C_VEL
LIN {X 0,Y 355.061,Z 388.579,A -85,B 0,C 180,E1 13199.336,E2 13199.336} C_VEL
LIN {X 0,Y 351.184,Z 419.833,A -85,B 0,C 180,E1 13201.68,E2 13201.68} C_VEL
LIN {X 0,Y 347.044,Z 447.803,A -85,B 0,C 180,E1 13204.883,E2 13204.883} C_VEL
LIN {X 0,Y 343.296,Z 472.992,A -85,B 0,C 180,E1 13209.074,E2 13209.074} C_VEL
LIN {X 0,Y 341.065,Z 493.202,A -85,B 0,C 180,E1 13213.946,E2 13213.946} C_VEL
LIN {X 0,Y 340.311,Z 507.652,A -85,B 0,C 180,E1 13219.137,E2 13219.137} C_VEL
LIN {X 0,Y 340.659,Z 515.474,A -85,B 0,C 180,E1 13223.641,E2 13223.641} C_VEL
LIN {X 0,Y 340.988,Z 518.966,A -85,B 0,C 180,E1 13227.463,E2 13227.463} C_VEL
LIN {X 0,Y 340.958,Z 519.058,A -85,B 0,C 180,E1 13232.536,E2 13232.536} C_VEL
LIN {X 0,Y 340.498,Z 514.168,A -85,B 0,C 180,E1 13237.639,E2 13237.639} C_VEL
LIN {X 0,Y 340.325,Z 504.05,A -85,B 0,C 180,E1 13242.808,E2 13242.808} C_VEL
LIN {X 0,Y 341.734,Z 488.142,A -85,B 0,C 180,E1 13248.004,E2 13248.004} C_VEL
LIN {X 0,Y 344.943,Z 466.401,A -85,B 0,C 180,E1 13252.845,E2 13252.845} C_VEL
LIN {X 0,Y 349.411,Z 440.99,A -85,B 0,C 180,E1 13256.792,E2 13256.792} C_VEL
LIN {X 0,Y 350.776,Z 433.111,A -85,B 0,C 180,E1 13257.761,E2 13257.761} C_VEL
LIN {X 0,Y 349.602,Z 419.269,A -85,B 0,C 180,E1 13259.52,E2 13259.52} C_VEL
LIN {X 0,Y 348.413,Z 404.6,A -85,B 0,C 180,E1 13261.078,E2 13261.078} C_VEL
LIN {X 0,Y 352.516,Z 374.131,A -85,B 0,C 180,E1 13263.003,E2 13263.003} C_VEL
LIN {X 0,Y 353.385,Z 354.568,A -85,B 0,C 180,E1 13263.845,E2 13263.845} C_VEL
LIN {X 0,Y 340.695,Z 321.301,A -85,B 0,C 180,E1 13266.192,E2 13266.192} C_VEL
LIN {X 0,Y 329.509,Z 299.393,A -85,B 0,C 180,E1 13268.231,E2 13268.231} C_VEL
LIN {X 0,Y 329.35,Z 297.81,A -85,B 0,C 180,E1 13268.42,E2 13268.42} C_VEL
LIN {X 0,Y 329.324,Z 297.81,A -85,B 0,C 180,E1 13273.417,E2 13273.417} C_VEL
LIN {X 0,Y 329.369,Z 297.81,A -85,B 0,C 180,E1 13281.154,E2 13281.154} C_VEL
LIN {X 0,Y 329.408,Z 297.81,A -85,B 0,C 180,E1 13286.671,E2 13286.671} C_VEL
LIN {X 0,Y 329.654,Z 297.81,A -85,B 0,C 180,E1 13292.775,E2 13292.775} C_VEL
LIN {X 0,Y 329.914,Z 297.81,A -85,B 0,C 180,E1 13298.553,E2 13298.553} C_VEL
LIN {X 0,Y 330.315,Z 297.81,A -85,B 0,C 180,E1 13306.812,E2 13306.812} C_VEL
LIN {X 0,Y 330.901,Z 297.81,A -85,B 0,C 180,E1 13314.783,E2 13314.783} C_VEL
LIN {X 0,Y 331.222,Z 297.81,A -85,B 0,C 180,E1 13320.016,E2 13320.016} C_VEL
LIN {X 0,Y 330.71,Z 297.81,A -85,B 0,C 180,E1 13327.884,E2 13327.884} C_VEL
LIN {X 0,Y 330.283,Z 297.81,A -85,B 0,C 180,E1 13335.928,E2 13335.928} C_VEL
LIN {X 0,Y 330.031,Z 297.81,A -85,B 0,C 180,E1 13341.826,E2 13341.826} C_VEL
LIN {X 0,Y 342.254,Z 328.351,A -85,B 0,C 180,E1 13344.955,E2 13344.955} C_VEL
LIN {X 0,Y 347.93,Z 353.058,A -85,B 0,C 180,E1 13347.809,E2 13347.809} C_VEL
LIN {X 0,Y 344.796,Z 376.968,A -85,B 0,C 180,E1 13350.693,E2 13350.693} C_VEL
LIN {X 0,Y 340.794,Z 397.32,A -85,B 0,C 180,E1 13354.364,E2 13354.364} C_VEL
LIN {X 0,Y 337.583,Z 411.76,A -85,B 0,C 180,E1 13358.385,E2 13358.385} C_VEL
LIN {X 0,Y 335.474,Z 420.666,A -85,B 0,C 180,E1 13362.456,E2 13362.456} C_VEL
LIN {X 0,Y 333.942,Z 425.429,A -85,B 0,C 180,E1 13367.328,E2 13367.328} C_VEL
LIN {X 0,Y 333.607,Z 424.638,A -85,B 0,C 180,E1 13371.79,E2 13371.79} C_VEL
LIN {X 0,Y 334.504,Z 418.178,A -85,B 0,C 180,E1 13376.617,E2 13376.617} C_VEL
LIN {X 0,Y 336.306,Z 405.967,A -85,B 0,C 180,E1 13381.195,E2 13381.195} C_VEL
LIN {X 0,Y 338.904,Z 388.364,A -85,B 0,C 180,E1 13385.256,E2 13385.256} C_VEL
LIN {X 0,Y 341.77,Z 366.709,A -85,B 0,C 180,E1 13388.561,E2 13388.561} C_VEL
LIN {X 0,Y 343.235,Z 346.358,A -85,B 0,C 180,E1 13390.748,E2 13390.748} C_VEL
LIN {X 0,Y 336.911,Z 318.929,A -85,B 0,C 180,E1 13393.243,E2 13393.243} C_VEL
LIN {X 0,Y 333.25,Z 308.494,A -85,B 0,C 180,E1 13394.124,E2 13394.124} C_VEL
LIN {X 0,Y 340.077,Z 335.346,A -85,B 0,C 180,E1 13395.533,E2 13395.533} C_VEL
LIN {X 0,Y 341.331,Z 350.373,A -85,B 0,C 180,E1 13396.648,E2 13396.648} C_VEL
LIN {X 0,Y 339.574,Z 373.201,A -85,B 0,C 180,E1 13398.952,E2 13398.952} C_VEL
LIN {X 0,Y 337.361,Z 394.062,A -85,B 0,C 180,E1 13402.289,E2 13402.289} C_VEL
LIN {X 0,Y 335.517,Z 409.353,A -85,B 0,C 180,E1 13406.132,E2 13406.132} C_VEL
LIN {X 0,Y 334.184,Z 419.974,A -85,B 0,C 180,E1 13410.648,E2 13410.648} C_VEL
LIN {X 0,Y 333.595,Z 424.747,A -85,B 0,C 180,E1 13415.455,E2 13415.455} C_VEL
LIN {X 0,Y 333.722,Z 424.916,A -85,B 0,C 180,E1 13417.797,E2 13417.797} C_VEL
LIN {X 0,Y 334.673,Z 421.985,A -85,B 0,C 180,E1 13421.707,E2 13421.707} C_VEL
LIN {X 0,Y 336.493,Z 413.138,A -85,B 0,C 180,E1 13426.278,E2 13426.278} C_VEL
LIN {X 0,Y 339.239,Z 398.233,A -85,B 0,C 180,E1 13430.506,E2 13430.506} C_VEL
LIN {X 0,Y 342.16,Z 379.058,A -85,B 0,C 180,E1 13433.893,E2 13433.893} C_VEL
LIN {X 0,Y 344.736,Z 356.675,A -85,B 0,C 180,E1 13436.413,E2 13436.413} C_VEL
LIN {X 0,Y 344.498,Z 344.443,A -85,B 0,C 180,E1 13437.463,E2 13437.463} C_VEL
LIN {X 0,Y 337.827,Z 319.679,A -85,B 0,C 180,E1 13439.301,E2 13439.301} C_VEL
LIN {X 0,Y 329.667,Z 297.81,A -85,B 0,C 180,E1 13440.708,E2 13440.708} C_VEL
LIN {X 0,Y 329.381,Z 297.81,A -85,B 0,C 180,E1 13448.819,E2 13448.819} C_VEL
LIN {X 0,Y 329.321,Z 297.81,A -85,B 0,C 180,E1 13456.557,E2 13456.557} C_VEL
LIN {X 0,Y 329.346,Z 297.81,A -85,B 0,C 180,E1 13463.42,E2 13463.42} C_VEL
LIN {X 0,Y 329.585,Z 297.81,A -85,B 0,C 180,E1 13470.45,E2 13470.45} C_VEL
LIN {X 0,Y 329.965,Z 297.81,A -85,B 0,C 180,E1 13478.521,E2 13478.521} C_VEL
LIN {X 0,Y 330.37,Z 297.81,A -85,B 0,C 180,E1 13486.781,E2 13486.781} C_VEL
LIN {X 0,Y 330.924,Z 297.81,A -85,B 0,C 180,E1 13494.751,E2 13494.751} C_VEL
LIN {X 0,Y 331.365,Z 297.81,A -85,B 0,C 180,E1 13499.984,E2 13499.984} C_VEL
LIN {X 0,Y 330.756,Z 297.81,A -85,B 0,C 180,E1 13507.85,E2 13507.85} C_VEL
LIN {X 0,Y 330.3,Z 297.81,A -85,B 0,C 180,E1 13515.893,E2 13515.893} C_VEL
LIN {X 0,Y 329.846,Z 297.81,A -85,B 0,C 180,E1 13524.297,E2 13524.297} C_VEL
LIN {X 0,Y 329.588,Z 297.81,A -85,B 0,C 180,E1 13530.222,E2 13530.222} C_VEL
LIN {X 0,Y 329.358,Z 297.81,A -85,B 0,C 180,E1 13536.537,E2 13536.537} C_VEL
LIN {X 0,Y 329.371,Z 297.81,A -85,B 0,C 180,E1 13543.389,E2 13543.389} C_VEL
LIN {X 0,Y 329.444,Z 297.81,A -85,B 0,C 180,E1 13551.115,E2 13551.115} C_VEL
LIN {X 0,Y 329.557,Z 297.81,A -85,B 0,C 180,E1 13554.308,E2 13554.308} C_VEL
LIN {X 0,Y 350.451,Z 356.625,A -85,B 0,C 180,E1 13557.431,E2 13557.431} C_VEL
LIN {X 0,Y 347.689,Z 389.032,A -85,B 0,C 180,E1 13558.885,E2 13558.885} C_VEL
LIN {X 0,Y 343.904,Z 418.476,A -85,B 0,C 180,E1 13561.14,E2 13561.14} C_VEL
LIN {X 0,Y 339.475,Z 447.218,A -85,B 0,C 180,E1 13564.492,E2 13564.492} C_VEL
LIN {X 0,Y 335.727,Z 471.326,A -85,B 0,C 180,E1 13568.58,E2 13568.58} C_VEL
LIN {X 0,Y 333.222,Z 491.77,A -85,B 0,C 180,E1 13573.558,E2 13573.558} C_VEL
LIN {X 0,Y 332.432,Z 506.495,A -85,B 0,C 180,E1 13578.929,E2 13578.929} C_VEL
LIN {X 0,Y 332.792,Z 514.289,A -85,B 0,C 180,E1 13583.49,E2 13583.49} C_VEL
LIN {X 0,Y 333.15,Z 517.831,A -85,B 0,C 180,E1 13587.403,E2 13587.403} C_VEL
LIN {X 0,Y 333.121,Z 517.969,A -85,B 0,C 180,E1 13592.596,E2 13592.596} C_VEL
LIN {X 0,Y 332.599,Z 513.087,A -85,B 0,C 180,E1 13597.822,E2 13597.822} C_VEL
LIN {X 0,Y 332.457,Z 502.995,A -85,B 0,C 180,E1 13603.117,E2 13603.117} C_VEL
LIN {X 0,Y 334.058,Z 486.872,A -85,B 0,C 180,E1 13608.495,E2 13608.495} C_VEL
LIN {X 0,Y 337.482,Z 465.404,A -85,B 0,C 180,E1 13613.379,E2 13613.379} C_VEL
LIN {X 0,Y 342.197,Z 440.084,A -85,B 0,C 180,E1 13617.389,E2 13617.389} C_VEL
LIN {X 0,Y 347.358,Z 411.308,A -85,B 0,C 180,E1 13620.512,E2 13620.512} C_VEL
LIN {X 0,Y 348.413,Z 404.6,A -85,B 0,C 180,E1 13621.078,E2 13621.078} C_VEL
LIN {X 0,Y 347.242,Z 389.309,A -85,B 0,C 180,E1 13622.485,E2 13622.485} C_VEL
LIN {X 0,Y 345.819,Z 373.514,A -85,B 0,C 180,E1 13623.705,E2 13623.705} C_VEL
LIN {X 0,Y 346.805,Z 357.014,A -85,B 0,C 180,E1 13624.446,E2 13624.446} C_VEL
LIN {X 0,Y 335.013,Z 325.466,A -85,B 0,C 180,E1 13626.801,E2 13626.801} C_VEL
LIN {X 0,Y 321.392,Z 297.81,A -85,B 0,C 180,E1 13629.543,E2 13629.543} C_VEL
LIN {X 0,Y 321.309,Z 297.81,A -85,B 0,C 180,E1 13635.236,E2 13635.236} C_VEL
LIN {X 0,Y 321.425,Z 297.81,A -85,B 0,C 180,E1 13642.948,E2 13642.948} C_VEL
LIN {X 0,Y 321.521,Z 297.81,A -85,B 0,C 180,E1 13648.937,E2 13648.937} C_VEL
LIN {X 0,Y 321.795,Z 297.81,A -85,B 0,C 180,E1 13655.054,E2 13655.054} C_VEL
LIN {X 0,Y 322.062,Z 297.81,A -85,B 0,C 180,E1 13660.871,E2 13660.871} C_VEL
LIN {X 0,Y 322.536,Z 297.81,A -85,B 0,C 180,E1 13669.259,E2 13669.259} C_VEL
LIN {X 0,Y 323.269,Z 297.81,A -85,B 0,C 180,E1 13677.341,E2 13677.341} C_VEL
LIN {X 0,Y 323.169,Z 297.81,A -85,B 0,C 180,E1 13682.693,E2 13682.693} C_VEL
LIN {X 0,Y 322.632,Z 297.81,A -85,B 0,C 180,E1 13690.831,E2 13690.831} C_VEL
LIN {X 0,Y 322.146,Z 297.81,A -85,B 0,C 180,E1 13699.159,E2 13699.159} C_VEL
LIN {X 0,Y 322.115,Z 298.638,A -85,B 0,C 180,E1 13700.743,E2 13700.743} C_VEL
LIN {X 0,Y 334.557,Z 327.718,A -85,B 0,C 180,E1 13703.968,E2 13703.968} C_VEL
LIN {X 0,Y 340.555,Z 352.39,A -85,B 0,C 180,E1 13706.911,E2 13706.911} C_VEL
LIN {X 0,Y 340.523,Z 362.691,A -85,B 0,C 180,E1 13708.145,E2 13708.145} C_VEL
LIN {X 0,Y 336.324,Z 385.278,A -85,B 0,C 180,E1 13711.288,E2 13711.288} C_VEL
LIN {X 0,Y 332.285,Z 403.7,A -85,B 0,C 180,E1 13715.173,E2 13715.173} C_VEL
LIN {X 0,Y 329.1,Z 416.691,A -85,B 0,C 180,E1 13719.504,E2 13719.504} C_VEL
LIN {X 0,Y 327.193,Z 424,A -85,B 0,C 180,E1 13723.797,E2 13723.797} C_VEL
LIN {X 0,Y 326.054,Z 426.696,A -85,B 0,C 180,E1 13727.8,E2 13727.8} C_VEL
LIN {X 0,Y 325.926,Z 424.683,A -85,B 0,C 180,E1 13732.996,E2 13732.996} C_VEL
LIN {X 0,Y 327.103,Z 416.693,A -85,B 0,C 180,E1 13737.938,E2 13737.938} C_VEL
LIN {X 0,Y 329.08,Z 403.971,A -85,B 0,C 180,E1 13742.272,E2 13742.272} C_VEL
LIN {X 0,Y 331.85,Z 385.602,A -85,B 0,C 180,E1 13746.263,E2 13746.263} C_VEL
LIN {X 0,Y 334.993,Z 362.627,A -85,B 0,C 180,E1 13749.569,E2 13749.569} C_VEL
LIN {X 0,Y 335.75,Z 347.822,A -85,B 0,C 180,E1 13751.154,E2 13751.154} C_VEL
LIN {X 0,Y 329.624,Z 320.759,A -85,B 0,C 180,E1 13753.72,E2 13753.72} C_VEL
LIN {X 0,Y 328.316,Z 317.899,A -85,B 0,C 180,E1 13753.993,E2 13753.993} C_VEL
LIN {X 0,Y 333.805,Z 343.853,A -85,B 0,C 180,E1 13755.663,E2 13755.663} C_VEL
LIN {X 0,Y 332.603,Z 367.753,A -85,B 0,C 180,E1 13757.822,E2 13757.822} C_VEL
LIN {X 0,Y 330.486,Z 388.703,A -85,B 0,C 180,E1 13760.805,E2 13760.805} C_VEL
LIN {X 0,Y 328.448,Z 405.215,A -85,B 0,C 180,E1 13764.398,E2 13764.398} C_VEL
LIN {X 0,Y 326.812,Z 417.497,A -85,B 0,C 180,E1 13768.678,E2 13768.678} C_VEL
LIN {X 0,Y 325.999,Z 423.829,A -85,B 0,C 180,E1 13772.654,E2 13772.654} C_VEL
LIN {X 0,Y 325.771,Z 425.756,A -85,B 0,C 180,E1 13775.316,E2 13775.316} C_VEL
LIN {X 0,Y 325.924,Z 425.971,A -85,B 0,C 180,E1 13777.985,E2 13777.985} C_VEL
LIN {X 0,Y 326.937,Z 422.954,A -85,B 0,C 180,E1 13781.988,E2 13781.988} C_VEL
LIN {X 0,Y 328.908,Z 413.993,A -85,B 0,C 180,E1 13786.664,E2 13786.664} C_VEL
LIN {X 0,Y 331.794,Z 399.135,A -85,B 0,C 180,E1 13790.938,E2 13790.938} C_VEL
LIN {X 0,Y 334.905,Z 379.723,A -85,B 0,C 180,E1 13794.416,E2 13794.416} C_VEL
LIN {X 0,Y 337.659,Z 356.705,A -85,B 0,C 180,E1 13797.018,E2 13797.018} C_VEL
LIN {X 0,Y 336.928,Z 344.168,A -85,B 0,C 180,E1 13798.133,E2 13798.133} C_VEL
LIN {X 0,Y 329.922,Z 319.237,A -85,B 0,C 180,E1 13800.014,E2 13800.014} C_VEL
LIN {X 0,Y 321.756,Z 297.81,A -85,B 0,C 180,E1 13801.451,E2 13801.451} C_VEL
LIN {X 0,Y 321.415,Z 297.81,A -85,B 0,C 180,E1 13807.614,E2 13807.614} C_VEL
LIN {X 0,Y 321.302,Z 297.81,A -85,B 0,C 180,E1 13815.187,E2 13815.187} C_VEL
LIN {X 0,Y 321.408,Z 297.81,A -85,B 0,C 180,E1 13822.954,E2 13822.954} C_VEL
LIN {X 0,Y 321.503,Z 297.81,A -85,B 0,C 180,E1 13828.895,E2 13828.895} C_VEL
LIN {X 0,Y 321.808,Z 297.81,A -85,B 0,C 180,E1 13835.018,E2 13835.018} C_VEL
LIN {X 0,Y 322.123,Z 297.81,A -85,B 0,C 180,E1 13840.839,E2 13840.839} C_VEL
LIN {X 0,Y 322.58,Z 297.81,A -85,B 0,C 180,E1 13849.225,E2 13849.225} C_VEL
LIN {X 0,Y 323.284,Z 297.81,A -85,B 0,C 180,E1 13857.308,E2 13857.308} C_VEL
LIN {X 0,Y 323.215,Z 297.81,A -85,B 0,C 180,E1 13862.659,E2 13862.659} C_VEL
LIN {X 0,Y 322.677,Z 297.81,A -85,B 0,C 180,E1 13870.865,E2 13870.865} C_VEL
LIN {X 0,Y 322.15,Z 297.81,A -85,B 0,C 180,E1 13879.124,E2 13879.124} C_VEL
LIN {X 0,Y 321.783,Z 297.81,A -85,B 0,C 180,E1 13886.999,E2 13886.999} C_VEL
LIN {X 0,Y 321.479,Z 297.81,A -85,B 0,C 180,E1 13894.263,E2 13894.263} C_VEL
LIN {X 0,Y 321.35,Z 297.81,A -85,B 0,C 180,E1 13901.293,E2 13901.293} C_VEL
LIN {X 0,Y 321.393,Z 297.81,A -85,B 0,C 180,E1 13908.903,E2 13908.903} C_VEL
LIN {X 0,Y 321.678,Z 298.27,A -85,B 0,C 180,E1 13913.64,E2 13913.64} C_VEL
LIN {X 0,Y 342.872,Z 356.675,A -85,B 0,C 180,E1 13916.866,E2 13916.866} C_VEL
LIN {X 0,Y 340.333,Z 389.394,A -85,B 0,C 180,E1 13918.415,E2 13918.415} C_VEL
LIN {X 0,Y 336.24,Z 419.553,A -85,B 0,C 180,E1 13920.821,E2 13920.821} C_VEL
LIN {X 0,Y 331.763,Z 447.54,A -85,B 0,C 180,E1 13924.218,E2 13924.218} C_VEL
LIN {X 0,Y 327.899,Z 471.307,A -85,B 0,C 180,E1 13928.397,E2 13928.397} C_VEL
LIN {X 0,Y 325.347,Z 491.498,A -85,B 0,C 180,E1 13933.512,E2 13933.512} C_VEL
LIN {X 0,Y 324.581,Z 504.535,A -85,B 0,C 180,E1 13938.333,E2 13938.333} C_VEL
LIN {X 0,Y 324.914,Z 513.093,A -85,B 0,C 180,E1 13943.332,E2 13943.332} C_VEL
LIN {X 0,Y 325.317,Z 516.686,A -85,B 0,C 180,E1 13947.341,E2 13947.341} C_VEL
LIN {X 0,Y 325.27,Z 516.876,A -85,B 0,C 180,E1 13952.658,E2 13952.658} C_VEL
LIN {X 0,Y 324.721,Z 512.015,A -85,B 0,C 180,E1 13958.013,E2 13958.013} C_VEL
LIN {X 0,Y 324.597,Z 501.94,A -85,B 0,C 180,E1 13963.44,E2 13963.44} C_VEL
LIN {X 0,Y 326.334,Z 486.073,A -85,B 0,C 180,E1 13968.885,E2 13968.885} C_VEL
LIN {X 0,Y 330.074,Z 464.469,A -85,B 0,C 180,E1 13973.924,E2 13973.924} C_VEL
LIN {X 0,Y 335.105,Z 438.84,A -85,B 0,C 180,E1 13978.068,E2 13978.068} C_VEL
LIN {X 0,Y 340.477,Z 410.414,A -85,B 0,C 180,E1 13981.197,E2 13981.197} C_VEL
LIN {X 0,Y 345.117,Z 379.644,A -85,B 0,C 180,E1 13983.382,E2 13983.382} C_VEL
LIN {X 0,Y 345.819,Z 373.514,A -85,B 0,C 180,E1 13983.705,E2 13983.705} C_VEL
LIN {X 0,Y 344.005,Z 361.622,A -85,B 0,C 180,E1 13984.562,E2 13984.562} C_VEL
LIN {X 0,Y 335.096,Z 343.373,A -85,B 0,C 180,E1 13986.302,E2 13986.302} C_VEL
LIN {X 0,Y 320.894,Z 312.75,A -85,B 0,C 180,E1 13989.112,E2 13989.112} C_VEL
LIN {X 0,Y 313.535,Z 299.022,A -85,B 0,C 180,E1 13990.677,E2 13990.677} C_VEL
LIN {X 0,Y 313.414,Z 297.81,A -85,B 0,C 180,E1 13990.742,E2 13990.742} C_VEL
LIN {X 0,Y 313.309,Z 297.81,A -85,B 0,C 180,E1 13997.623,E2 13997.623} C_VEL
LIN {X 0,Y 313.495,Z 297.81,A -85,B 0,C 180,E1 14004.913,E2 14004.913} C_VEL
LIN {X 0,Y 313.669,Z 297.81,A -85,B 0,C 180,E1 14011.263,E2 14011.263} C_VEL
LIN {X 0,Y 313.967,Z 297.81,A -85,B 0,C 180,E1 14017.405,E2 14017.405} C_VEL
LIN {X 0,Y 314.323,Z 297.81,A -85,B 0,C 180,E1 14023.769,E2 14023.769} C_VEL
LIN {X 0,Y 314.82,Z 297.81,A -85,B 0,C 180,E1 14031.749,E2 14031.749} C_VEL
LIN {X 0,Y 315.363,Z 297.81,A -85,B 0,C 180,E1 14037.274,E2 14037.274} C_VEL
LIN {X 0,Y 315.28,Z 297.81,A -85,B 0,C 180,E1 14042.761,E2 14042.761} C_VEL
LIN {X 0,Y 314.715,Z 297.81,A -85,B 0,C 180,E1 14051.075,E2 14051.075} C_VEL
LIN {X 0,Y 314.261,Z 297.81,A -85,B 0,C 180,E1 14059.295,E2 14059.295} C_VEL
LIN {X 0,Y 314.594,Z 300.171,A -85,B 0,C 180,E1 14059.638,E2 14059.638} C_VEL
LIN {X 0,Y 326.058,Z 324.878,A -85,B 0,C 180,E1 14062.644,E2 14062.644} C_VEL
LIN {X 0,Y 332.743,Z 349.298,A -85,B 0,C 180,E1 14065.657,E2 14065.657} C_VEL
LIN {X 0,Y 333.942,Z 361.858,A -85,B 0,C 180,E1 14067.286,E2 14067.286} C_VEL
LIN {X 0,Y 329.494,Z 385.187,A -85,B 0,C 180,E1 14070.505,E2 14070.505} C_VEL
LIN {X 0,Y 325.198,Z 403.675,A -85,B 0,C 180,E1 14074.402,E2 14074.402} C_VEL
LIN {X 0,Y 321.84,Z 416.694,A -85,B 0,C 180,E1 14078.654,E2 14078.654} C_VEL
LIN {X 0,Y 319.452,Z 425.215,A -85,B 0,C 180,E1 14083.621,E2 14083.621} C_VEL
LIN {X 0,Y 318.04,Z 427.859,A -85,B 0,C 180,E1 14089.417,E2 14089.417} C_VEL
LIN {X 0,Y 318.315,Z 423.972,A -85,B 0,C 180,E1 14094.558,E2 14094.558} C_VEL
LIN {X 0,Y 319.834,Z 414.635,A -85,B 0,C 180,E1 14099.386,E2 14099.386} C_VEL
LIN {X 0,Y 322.219,Z 399.807,A -85,B 0,C 180,E1 14103.854,E2 14103.854} C_VEL
LIN {X 0,Y 325.417,Z 379.338,A -85,B 0,C 180,E1 14107.84,E2 14107.84} C_VEL
LIN {X 0,Y 328.693,Z 354.506,A -85,B 0,C 180,E1 14110.995,E2 14110.995} C_VEL
LIN {X 0,Y 324.284,Z 329.645,A -85,B 0,C 180,E1 14113.592,E2 14113.592} C_VEL
LIN {X 0,Y 322.872,Z 327.201,A -85,B 0,C 180,E1 14113.994,E2 14113.994} C_VEL
LIN {X 0,Y 326.599,Z 349.439,A -85,B 0,C 180,E1 14115.603,E2 14115.603} C_VEL
LIN {X 0,Y 324.626,Z 373.729,A -85,B 0,C 180,E1 14118.047,E2 14118.047} C_VEL
LIN {X 0,Y 322.378,Z 393.758,A -85,B 0,C 180,E1 14121.251,E2 14121.251} C_VEL
LIN {X 0,Y 320.234,Z 409.972,A -85,B 0,C 180,E1 14125.271,E2 14125.271} C_VEL
LIN {X 0,Y 318.63,Z 421.321,A -85,B 0,C 180,E1 14130.001,E2 14130.001} C_VEL
LIN {X 0,Y 317.976,Z 426.422,A -85,B 0,C 180,E1 14134.505,E2 14134.505} C_VEL
LIN {X 0,Y 318.128,Z 427.022,A -85,B 0,C 180,E1 14138.182,E2 14138.182} C_VEL
LIN {X 0,Y 319.229,Z 423.916,A -85,B 0,C 180,E1 14142.282,E2 14142.282} C_VEL
LIN {X 0,Y 321.359,Z 414.835,A -85,B 0,C 180,E1 14147.067,E2 14147.067} C_VEL
LIN {X 0,Y 324.149,Z 401.107,A -85,B 0,C 180,E1 14151.137,E2 14151.137} C_VEL
LIN {X 0,Y 327.216,Z 383.307,A -85,B 0,C 180,E1 14154.523,E2 14154.523} C_VEL
LIN {X 0,Y 330.256,Z 360.393,A -85,B 0,C 180,E1 14157.313,E2 14157.313} C_VEL
LIN {X 0,Y 330.279,Z 348.774,A -85,B 0,C 180,E1 14158.379,E2 14158.379} C_VEL
LIN {X 0,Y 324.129,Z 324.74,A -85,B 0,C 180,E1 14160.366,E2 14160.366} C_VEL
LIN {X 0,Y 313.72,Z 297.81,A -85,B 0,C 180,E1 14162.271,E2 14162.271} C_VEL
LIN {X 0,Y 313.339,Z 297.81,A -85,B 0,C 180,E1 14169.569,E2 14169.569} C_VEL
LIN {X 0,Y 313.298,Z 297.81,A -85,B 0,C 180,E1 14177.575,E2 14177.575} C_VEL
LIN {X 0,Y 313.495,Z 297.81,A -85,B 0,C 180,E1 14184.915,E2 14184.915} C_VEL
LIN {X 0,Y 313.636,Z 297.81,A -85,B 0,C 180,E1 14191.22,E2 14191.22} C_VEL
LIN {X 0,Y 314.011,Z 297.81,A -85,B 0,C 180,E1 14197.371,E2 14197.371} C_VEL
LIN {X 0,Y 314.372,Z 297.81,A -85,B 0,C 180,E1 14203.744,E2 14203.744} C_VEL
LIN {X 0,Y 314.855,Z 297.81,A -85,B 0,C 180,E1 14211.716,E2 14211.716} C_VEL
LIN {X 0,Y 315.567,Z 297.81,A -85,B 0,C 180,E1 14219.983,E2 14219.983} C_VEL
LIN {X 0,Y 314.9,Z 297.81,A -85,B 0,C 180,E1 14228.248,E2 14228.248} C_VEL
LIN {X 0,Y 314.453,Z 297.81,A -85,B 0,C 180,E1 14236.306,E2 14236.306} C_VEL
LIN {X 0,Y 313.913,Z 297.81,A -85,B 0,C 180,E1 14244.027,E2 14244.027} C_VEL
LIN {X 0,Y 313.615,Z 297.81,A -85,B 0,C 180,E1 14251.938,E2 14251.938} C_VEL
LIN {X 0,Y 313.342,Z 297.81,A -85,B 0,C 180,E1 14259.597,E2 14259.597} C_VEL
LIN {X 0,Y 313.361,Z 297.81,A -85,B 0,C 180,E1 14267.609,E2 14267.609} C_VEL
LIN {X 0,Y 313.681,Z 297.81,A -85,B 0,C 180,E1 14272.859,E2 14272.859} C_VEL
LIN {X 0,Y 335.042,Z 356.433,A -85,B 0,C 180,E1 14276.252,E2 14276.252} C_VEL
LIN {X 0,Y 335.04,Z 369.778,A -85,B 0,C 180,E1 14276.844,E2 14276.844} C_VEL
LIN {X 0,Y 331.323,Z 401.928,A -85,B 0,C 180,E1 14278.796,E2 14278.796} C_VEL
LIN {X 0,Y 326.84,Z 431.045,A -85,B 0,C 180,E1 14281.66,E2 14281.66} C_VEL
LIN {X 0,Y 322.244,Z 458.239,A -85,B 0,C 180,E1 14285.651,E2 14285.651} C_VEL
LIN {X 0,Y 318.733,Z 480.06,A -85,B 0,C 180,E1 14290.285,E2 14290.285} C_VEL
LIN {X 0,Y 316.986,Z 497.138,A -85,B 0,C 180,E1 14295.526,E2 14295.526} C_VEL
LIN {X 0,Y 316.828,Z 508.97,A -85,B 0,C 180,E1 14301.094,E2 14301.094} C_VEL
LIN {X 0,Y 317.365,Z 515.099,A -85,B 0,C 180,E1 14306.597,E2 14306.597} C_VEL
LIN {X 0,Y 317.611,Z 516.29,A -85,B 0,C 180,E1 14309.999,E2 14309.999} C_VEL
LIN {X 0,Y 317.153,Z 514.034,A -85,B 0,C 180,E1 14315.46,E2 14315.46} C_VEL
LIN {X 0,Y 316.61,Z 506.581,A -85,B 0,C 180,E1 14320.99,E2 14320.99} C_VEL
LIN {X 0,Y 317.443,Z 493.801,A -85,B 0,C 180,E1 14326.571,E2 14326.571} C_VEL
LIN {X 0,Y 320.483,Z 474.491,A -85,B 0,C 180,E1 14332.127,E2 14332.127} C_VEL
LIN {X 0,Y 325.412,Z 450.369,A -85,B 0,C 180,E1 14336.879,E2 14336.879} C_VEL
LIN {X 0,Y 331.142,Z 422.298,A -85,B 0,C 180,E1 14340.65,E2 14340.65} C_VEL
LIN {X 0,Y 336.675,Z 391.259,A -85,B 0,C 180,E1 14343.37,E2 14343.37} C_VEL
LIN {X 0,Y 340.135,Z 359.142,A -85,B 0,C 180,E1 14345.088,E2 14345.088} C_VEL
LIN {X 0,Y 335.096,Z 343.373,A -85,B 0,C 180,E1 14346.302,E2 14346.302} C_VEL
LIN {X 0,Y 328.77,Z 333.813,A -85,B 0,C 180,E1 14347.409,E2 14347.409} C_VEL
LIN {X 0,Y 316.786,Z 319.515,A -85,B 0,C 180,E1 14349.541,E2 14349.541} C_VEL
LIN {X 0,Y 305.449,Z 298.377,A -85,B 0,C 180,E1 14352.116,E2 14352.116} C_VEL
LIN {X 0,Y 305.387,Z 297.81,A -85,B 0,C 180,E1 14360.053,E2 14360.053} C_VEL
LIN {X 0,Y 305.57,Z 297.81,A -85,B 0,C 180,E1 14367.117,E2 14367.117} C_VEL
LIN {X 0,Y 305.825,Z 297.81,A -85,B 0,C 180,E1 14373.655,E2 14373.655} C_VEL
LIN {X 0,Y 306.121,Z 297.81,A -85,B 0,C 180,E1 14379.833,E2 14379.833} C_VEL
LIN {X 0,Y 306.48,Z 297.81,A -85,B 0,C 180,E1 14385.766,E2 14385.766} C_VEL
LIN {X 0,Y 307.115,Z 297.81,A -85,B 0,C 180,E1 14394.378,E2 14394.378} C_VEL
LIN {X 0,Y 307.524,Z 297.81,A -85,B 0,C 180,E1 14400.018,E2 14400.018} C_VEL
LIN {X 0,Y 306.92,Z 297.81,A -85,B 0,C 180,E1 14408.5,E2 14408.5} C_VEL
LIN {X 0,Y 306.59,Z 297.81,A -85,B 0,C 180,E1 14414.265,E2 14414.265} C_VEL
LIN {X 0,Y 306.345,Z 297.952,A -85,B 0,C 180,E1 14418.135,E2 14418.135} C_VEL
LIN {X 0,Y 311.102,Z 308.257,A -85,B 0,C 180,E1 14419.407,E2 14419.407} C_VEL
LIN {X 0,Y 321.474,Z 333.108,A -85,B 0,C 180,E1 14422.621,E2 14422.621} C_VEL
LIN {X 0,Y 326.85,Z 357.431,A -85,B 0,C 180,E1 14425.85,E2 14425.85} C_VEL
LIN {X 0,Y 326.287,Z 367.845,A -85,B 0,C 180,E1 14427.194,E2 14427.194} C_VEL
LIN {X 0,Y 321.408,Z 390.806,A -85,B 0,C 180,E1 14430.723,E2 14430.723} C_VEL
LIN {X 0,Y 317.011,Z 408.238,A -85,B 0,C 180,E1 14434.857,E2 14434.857} C_VEL
LIN {X 0,Y 313.476,Z 420.768,A -85,B 0,C 180,E1 14439.629,E2 14439.629} C_VEL
LIN {X 0,Y 311.737,Z 426.43,A -85,B 0,C 180,E1 14443.441,E2 14443.441} C_VEL
LIN {X 0,Y 310.554,Z 428.869,A -85,B 0,C 180,E1 14447.137,E2 14447.137} C_VEL
LIN {X 0,Y 310.209,Z 427.188,A -85,B 0,C 180,E1 14452.675,E2 14452.675} C_VEL
LIN {X 0,Y 311.412,Z 419.718,A -85,B 0,C 180,E1 14457.791,E2 14457.791} C_VEL
LIN {X 0,Y 313.499,Z 407.184,A -85,B 0,C 180,E1 14462.437,E2 14462.437} C_VEL
LIN {X 0,Y 316.378,Z 389.987,A -85,B 0,C 180,E1 14466.527,E2 14466.527} C_VEL
LIN {X 0,Y 319.806,Z 366.975,A -85,B 0,C 180,E1 14470.144,E2 14470.144} C_VEL
LIN {X 0,Y 321.096,Z 352.072,A -85,B 0,C 180,E1 14471.861,E2 14471.861} C_VEL
LIN {X 0,Y 317.244,Z 335.027,A -85,B 0,C 180,E1 14473.773,E2 14473.773} C_VEL
LIN {X 0,Y 316.941,Z 335.477,A -85,B 0,C 180,E1 14473.979,E2 14473.979} C_VEL
LIN {X 0,Y 319.061,Z 351.842,A -85,B 0,C 180,E1 14475.274,E2 14475.274} C_VEL
LIN {X 0,Y 317.043,Z 375.471,A -85,B 0,C 180,E1 14477.757,E2 14477.757} C_VEL
LIN {X 0,Y 314.676,Z 395.265,A -85,B 0,C 180,E1 14481.035,E2 14481.035} C_VEL
LIN {X 0,Y 312.485,Z 411.313,A -85,B 0,C 180,E1 14485.153,E2 14485.153} C_VEL
LIN {X 0,Y 310.82,Z 422.541,A -85,B 0,C 180,E1 14490.001,E2 14490.001} C_VEL
LIN {X 0,Y 310.333,Z 426.177,A -85,B 0,C 180,E1 14492.788,E2 14492.788} C_VEL
LIN {X 0,Y 310.134,Z 427.985,A -85,B 0,C 180,E1 14495.585,E2 14495.585} C_VEL
LIN {X 0,Y 310.336,Z 428.073,A -85,B 0,C 180,E1 14498.389,E2 14498.389} C_VEL
LIN {X 0,Y 311.528,Z 424.878,A -85,B 0,C 180,E1 14502.591,E2 14502.591} C_VEL
LIN {X 0,Y 313.822,Z 415.672,A -85,B 0,C 180,E1 14507.49,E2 14507.49} C_VEL
LIN {X 0,Y 316.768,Z 401.823,A -85,B 0,C 180,E1 14511.654,E2 14511.654} C_VEL
LIN {X 0,Y 320.028,Z 383.804,A -85,B 0,C 180,E1 14515.112,E2 14515.112} C_VEL
LIN {X 0,Y 323.094,Z 361.737,A -85,B 0,C 180,E1 14517.844,E2 14517.844} C_VEL
LIN {X 0,Y 322.756,Z 348.396,A -85,B 0,C 180,E1 14519.121,E2 14519.121} C_VEL
LIN {X 0,Y 316.252,Z 324.356,A -85,B 0,C 180,E1 14521.142,E2 14521.142} C_VEL
LIN {X 0,Y 305.726,Z 297.81,A -85,B 0,C 180,E1 14523.061,E2 14523.061} C_VEL
LIN {X 0,Y 305.375,Z 297.81,A -85,B 0,C 180,E1 14532.136,E2 14532.136} C_VEL
LIN {X 0,Y 305.374,Z 297.81,A -85,B 0,C 180,E1 14540.005,E2 14540.005} C_VEL
LIN {X 0,Y 305.552,Z 297.81,A -85,B 0,C 180,E1 14547.095,E2 14547.095} C_VEL
LIN {X 0,Y 305.812,Z 297.81,A -85,B 0,C 180,E1 14553.614,E2 14553.614} C_VEL
LIN {X 0,Y 306.184,Z 297.81,A -85,B 0,C 180,E1 14559.799,E2 14559.799} C_VEL
LIN {X 0,Y 306.535,Z 297.81,A -85,B 0,C 180,E1 14565.732,E2 14565.732} C_VEL
LIN {X 0,Y 307.14,Z 297.81,A -85,B 0,C 180,E1 14574.343,E2 14574.343} C_VEL
LIN {X 0,Y 307.662,Z 297.81,A -85,B 0,C 180,E1 14579.982,E2 14579.982} C_VEL
LIN {X 0,Y 306.961,Z 297.81,A -85,B 0,C 180,E1 14588.463,E2 14588.463} C_VEL
LIN {X 0,Y 306.641,Z 297.81,A -85,B 0,C 180,E1 14594.226,E2 14594.226} C_VEL
LIN {X 0,Y 306.053,Z 297.81,A -85,B 0,C 180,E1 14603.213,E2 14603.213} C_VEL
LIN {X 0,Y 305.745,Z 297.81,A -85,B 0,C 180,E1 14609.555,E2 14609.555} C_VEL
LIN {X 0,Y 305.385,Z 297.81,A -85,B 0,C 180,E1 14617.756,E2 14617.756} C_VEL
LIN {X 0,Y 305.456,Z 297.81,A -85,B 0,C 180,E1 14623.736,E2 14623.736} C_VEL
LIN {X 0,Y 305.677,Z 297.81,A -85,B 0,C 180,E1 14632.056,E2 14632.056} C_VEL
LIN {X 0,Y 326.977,Z 355.362,A -85,B 0,C 180,E1 14635.555,E2 14635.555} C_VEL
LIN {X 0,Y 328.366,Z 363.396,A -85,B 0,C 180,E1 14636.011,E2 14636.011} C_VEL
LIN {X 0,Y 324.827,Z 395.511,A -85,B 0,C 180,E1 14637.805,E2 14637.805} C_VEL
LIN {X 0,Y 320.316,Z 425.328,A -85,B 0,C 180,E1 14640.576,E2 14640.576} C_VEL
LIN {X 0,Y 315.609,Z 452.222,A -85,B 0,C 180,E1 14644.322,E2 14644.322} C_VEL
LIN {X 0,Y 311.534,Z 475.658,A -85,B 0,C 180,E1 14649.069,E2 14649.069} C_VEL
LIN {X 0,Y 309.399,Z 493.832,A -85,B 0,C 180,E1 14654.439,E2 14654.439} C_VEL
LIN {X 0,Y 308.922,Z 506.506,A -85,B 0,C 180,E1 14660.155,E2 14660.155} C_VEL
LIN {X 0,Y 309.435,Z 513.486,A -85,B 0,C 180,E1 14665.804,E2 14665.804} C_VEL
LIN {X 0,Y 309.797,Z 515.178,A -85,B 0,C 180,E1 14669.999,E2 14669.999} C_VEL
LIN {X 0,Y 309.3,Z 512.951,A -85,B 0,C 180,E1 14675.599,E2 14675.599} C_VEL
LIN {X 0,Y 308.728,Z 505.539,A -85,B 0,C 180,E1 14681.274,E2 14681.274} C_VEL
LIN {X 0,Y 309.839,Z 491.472,A -85,B 0,C 180,E1 14687.454,E2 14687.454} C_VEL
LIN {X 0,Y 313.285,Z 471.849,A -85,B 0,C 180,E1 14693.092,E2 14693.092} C_VEL
LIN {X 0,Y 318.717,Z 447.375,A -85,B 0,C 180,E1 14697.874,E2 14697.874} C_VEL
LIN {X 0,Y 324.647,Z 420.09,A -85,B 0,C 180,E1 14701.527,E2 14701.527} C_VEL
LIN {X 0,Y 330.302,Z 389.207,A -85,B 0,C 180,E1 14704.225,E2 14704.225} C_VEL
LIN {X 0,Y 333.47,Z 361.235,A -85,B 0,C 180,E1 14705.761,E2 14705.761} C_VEL
LIN {X 0,Y 323.593,Z 333.373,A -85,B 0,C 180,E1 14708.124,E2 14708.124} C_VEL
LIN {X 0,Y 316.786,Z 319.515,A -85,B 0,C 180,E1 14709.541,E2 14709.541} C_VEL
LIN {X 0,Y 309.921,Z 313.331,A -85,B 0,C 180,E1 14710.848,E2 14710.848} C_VEL
LIN {X 0,Y 302.51,Z 308.079,A -85,B 0,C 180,E1 14712.331,E2 14712.331} C_VEL
LIN {X 0,Y 297.52,Z 298.327,A -85,B 0,C 180,E1 14713.649,E2 14713.649} C_VEL
LIN {X 0,Y 297.447,Z 297.81,A -85,B 0,C 180,E1 14719.549,E2 14719.549} C_VEL
LIN {X 0,Y 297.54,Z 297.81,A -85,B 0,C 180,E1 14726.112,E2 14726.112} C_VEL
LIN {X 0,Y 297.853,Z 297.81,A -85,B 0,C 180,E1 14732.893,E2 14732.893} C_VEL
LIN {X 0,Y 298.163,Z 297.81,A -85,B 0,C 180,E1 14739.27,E2 14739.27} C_VEL
LIN {X 0,Y 298.504,Z 297.81,A -85,B 0,C 180,E1 14745.377,E2 14745.377} C_VEL
LIN {X 0,Y 299.179,Z 297.81,A -85,B 0,C 180,E1 14754.228,E2 14754.228} C_VEL
LIN {X 0,Y 299.634,Z 297.81,A -85,B 0,C 180,E1 14760.018,E2 14760.018} C_VEL
LIN {X 0,Y 298.997,Z 297.81,A -85,B 0,C 180,E1 14768.727,E2 14768.727} C_VEL
LIN {X 0,Y 298.482,Z 297.832,A -85,B 0,C 180,E1 14776.641,E2 14776.641} C_VEL
LIN {X 0,Y 301.04,Z 303.604,A -85,B 0,C 180,E1 14777.405,E2 14777.405} C_VEL
LIN {X 0,Y 313.011,Z 329.748,A -85,B 0,C 180,E1 14781.07,E2 14781.07} C_VEL
LIN {X 0,Y 319.308,Z 354.199,A -85,B 0,C 180,E1 14784.445,E2 14784.445} C_VEL
LIN {X 0,Y 320.032,Z 366.601,A -85,B 0,C 180,E1 14786.196,E2 14786.196} C_VEL
LIN {X 0,Y 314.803,Z 390.264,A -85,B 0,C 180,E1 14789.791,E2 14789.791} C_VEL
LIN {X 0,Y 309.908,Z 408.674,A -85,B 0,C 180,E1 14794.132,E2 14794.132} C_VEL
LIN {X 0,Y 306.006,Z 421.638,A -85,B 0,C 180,E1 14799.099,E2 14799.099} C_VEL
LIN {X 0,Y 303.644,Z 428.472,A -85,B 0,C 180,E1 14804.113,E2 14804.113} C_VEL
LIN {X 0,Y 302.387,Z 430.001,A -85,B 0,C 180,E1 14809.555,E2 14809.555} C_VEL
LIN {X 0,Y 302.666,Z 426.166,A -85,B 0,C 180,E1 14814.63,E2 14814.63} C_VEL
LIN {X 0,Y 304.205,Z 417.222,A -85,B 0,C 180,E1 14819.534,E2 14819.534} C_VEL
LIN {X 0,Y 306.783,Z 402.595,A -85,B 0,C 180,E1 14824.259,E2 14824.259} C_VEL
LIN {X 0,Y 310.202,Z 382.432,A -85,B 0,C 180,E1 14828.447,E2 14828.447} C_VEL
LIN {X 0,Y 313.795,Z 357.921,A -85,B 0,C 180,E1 14831.786,E2 14831.786} C_VEL
LIN {X 0,Y 311.913,Z 343.502,A -85,B 0,C 180,E1 14833.488,E2 14833.488} C_VEL
LIN {X 0,Y 310.451,Z 341.493,A -85,B 0,C 180,E1 14833.862,E2 14833.862} C_VEL
LIN {X 0,Y 311.456,Z 355.921,A -85,B 0,C 180,E1 14835.086,E2 14835.086} C_VEL
LIN {X 0,Y 309.176,Z 379.173,A -85,B 0,C 180,E1 14837.731,E2 14837.731} C_VEL
LIN {X 0,Y 306.758,Z 398.415,A -85,B 0,C 180,E1 14841.158,E2 14841.158} C_VEL
LIN {X 0,Y 304.526,Z 413.702,A -85,B 0,C 180,E1 14845.382,E2 14845.382} C_VEL
LIN {X 0,Y 302.996,Z 423.762,A -85,B 0,C 180,E1 14850.001,E2 14850.001} C_VEL
LIN {X 0,Y 302.42,Z 427.749,A -85,B 0,C 180,E1 14853.349,E2 14853.349} C_VEL
LIN {X 0,Y 302.549,Z 429.125,A -85,B 0,C 180,E1 14858.606,E2 14858.606} C_VEL
LIN {X 0,Y 304.091,Z 424.921,A -85,B 0,C 180,E1 14863.634,E2 14863.634} C_VEL
LIN {X 0,Y 306.744,Z 414.631,A -85,B 0,C 180,E1 14868.649,E2 14868.649} C_VEL
LIN {X 0,Y 310.067,Z 399.418,A -85,B 0,C 180,E1 14872.914,E2 14872.914} C_VEL
LIN {X 0,Y 313.616,Z 379.868,A -85,B 0,C 180,E1 14876.386,E2 14876.386} C_VEL
LIN {X 0,Y 316.566,Z 356.628,A -85,B 0,C 180,E1 14879.005,E2 14879.005} C_VEL
LIN {X 0,Y 311.642,Z 333.558,A -85,B 0,C 180,E1 14881.212,E2 14881.212} C_VEL
LIN {X 0,Y 297.745,Z 297.81,A -85,B 0,C 180,E1 14883.883,E2 14883.883} C_VEL
LIN {X 0,Y 297.442,Z 297.81,A -85,B 0,C 180,E1 14891.264,E2 14891.264} C_VEL
LIN {X 0,Y 297.451,Z 297.81,A -85,B 0,C 180,E1 14899.55,E2 14899.55} C_VEL
LIN {X 0,Y 297.502,Z 297.81,A -85,B 0,C 180,E1 14906.063,E2 14906.063} C_VEL
LIN {X 0,Y 297.839,Z 297.81,A -85,B 0,C 180,E1 14912.851,E2 14912.851} C_VEL
LIN {X 0,Y 298.222,Z 297.81,A -85,B 0,C 180,E1 14919.236,E2 14919.236} C_VEL
LIN {X 0,Y 298.56,Z 297.81,A -85,B 0,C 180,E1 14925.343,E2 14925.343} C_VEL
LIN {X 0,Y 299.204,Z 297.81,A -85,B 0,C 180,E1 14934.193,E2 14934.193} C_VEL
LIN {X 0,Y 299.756,Z 297.81,A -85,B 0,C 180,E1 14939.982,E2 14939.982} C_VEL
LIN {X 0,Y 299.039,Z 297.81,A -85,B 0,C 180,E1 14948.689,E2 14948.689} C_VEL
LIN {X 0,Y 298.504,Z 297.81,A -85,B 0,C 180,E1 14956.157,E2 14956.157} C_VEL
LIN {X 0,Y 297.985,Z 297.81,A -85,B 0,C 180,E1 14964.282,E2 14964.282} C_VEL
LIN {X 0,Y 297.719,Z 297.81,A -85,B 0,C 180,E1 14970.496,E2 14970.496} C_VEL
LIN {X 0,Y 297.482,Z 297.81,A -85,B 0,C 180,E1 14977.475,E2 14977.475} C_VEL
LIN {X 0,Y 297.509,Z 297.81,A -85,B 0,C 180,E1 14985.219,E2 14985.219} C_VEL
LIN {X 0,Y 297.67,Z 297.868,A -85,B 0,C 180,E1 14991.27,E2 14991.27} C_VEL
LIN {X 0,Y 318.479,Z 353.041,A -85,B 0,C 180,E1 14994.755,E2 14994.755} C_VEL
LIN {X 0,Y 321.075,Z 365.105,A -85,B 0,C 180,E1 14995.496,E2 14995.496} C_VEL
LIN {X 0,Y 317.296,Z 397.063,A -85,B 0,C 180,E1 14997.393,E2 14997.393} C_VEL
LIN {X 0,Y 312.493,Z 427.027,A -85,B 0,C 180,E1 15000.334,E2 15000.334} C_VEL
LIN {X 0,Y 307.698,Z 453.288,A -85,B 0,C 180,E1 15004.2,E2 15004.2} C_VEL
LIN {X 0,Y 303.709,Z 475.438,A -85,B 0,C 180,E1 15008.885,E2 15008.885} C_VEL
LIN {X 0,Y 301.597,Z 492.36,A -85,B 0,C 180,E1 15014.026,E2 15014.026} C_VEL
LIN {X 0,Y 301.046,Z 505.211,A -85,B 0,C 180,E1 15019.895,E2 15019.895} C_VEL
LIN {X 0,Y 301.596,Z 512.299,A -85,B 0,C 180,E1 15025.695,E2 15025.695} C_VEL
